(* Init ST03_125_F1 Absicherung Roboter iO (DigIn) *)
ST03_125_F1.sInit.InstName               :='ST03_125_F1';
ST03_125_F1.sInit.Description            :='Absicherung Roboter iO';
ST03_125_F1.sInit.BitInName              :='+3-125_F1';
ST03_125_F1.sInit.HomePosSignal          :=2; (* 0: Signal=Low, 1: Signal=High, 2: always  *)
ST03_125_F1.sInit.MaxTime                :=10;
ST03_125_F1.sInit.EnableInEveryMode       :=TRUE;

(* Init ST03_400_B12_6 Schwenkmodul GST (Roboterkopf) (DigIn) *)
ST03_400_B12_6.sInit.InstName           :='ST03_400_B12_6';
ST03_400_B12_6.sInit.Description        :='Rob. ST03 Schwenken GST';
ST03_400_B12_6.sInit.BitInName          :='+3-400_B12_6';
ST03_400_B12_6.sInit.HomePosSignal      :=2; (* 0: Signal=Low, 1: Signal=High, 2: always  *)
ST03_400_B12_6.sInit.MaxTime            :=2000;

(* Init ST03_400_B12_7 Schwenkmodul AST (Roboter) (DigIn) *)
ST03_400_B12_7.sInit.InstName           :='ST03_400_B12_7';
ST03_400_B12_7.sInit.Description        :='Rob. ST03 Schwenken AST';
ST03_400_B12_7.sInit.BitInName          :='+3-400_B12_7';
ST03_400_B12_7.sInit.HomePosSignal      :=2; (* 0: Signal=Low, 1: Signal=High, 2: always  *)
ST03_400_B12_7.sInit.MaxTime            :=2000;

(* Init St03_120_A1_A14 Rob. opt. Tool 2 ist Ein (DigIn) *)
St03_120_A1_A14.sInit.InstName           :='St03_120_A1_A14';
St03_120_A1_A14.sInit.Description        :='Rob. opt. Tool 2 ist Ein';
St03_120_A1_A14.sInit.BitInName          :='+3-120_A1_A14';
St03_120_A1_A14.sInit.HomePosSignal      :=2; (* 0: Signal=Low, 1: Signal=High, 2: always  *)
St03_120_A1_A14.sInit.MaxTime            :=2000;

(* Init ST03_BG3_S53_0 Start Band für Dummyprüfung (DigIn) *)
ST03_BG3_S53_0.sInit.InstName               :='ST03_BG3_S53_0';
ST03_BG3_S53_0.sInit.Description            :='Start Band für Dummyprüfung';
ST03_BG3_S53_0.sInit.BitInName              :='+0-BG3_S53_0';
ST03_BG3_S53_0.sInit.HomePosSignal          :=2; (* 0: Signal=Low, 1: Signal=High, 2: always  *)
ST03_BG3_S53_0.sInit.MaxTime                :=2000;
ST03_BG3_S53_0.sInit.EnableInEveryMode   	 :=TRUE;

(* Init ST03_BG3_X53_0 LED TasterStart Band für Dummyprüfung (DigOutIn) *)
ST03_BG3_X53_0.sInit.InstName          :='ST03_BG3_X53_0';
ST03_BG3_X53_0.sInit.Description       :='LED TasterStart Band für Dummyprüfung';
ST03_BG3_X53_0.sInit.BitOutName        :='+ST03_BG3_X53_0';
ST03_BG3_X53_0.sInit.BitInName         :='';
ST03_BG3_X53_0.sInit.HomePosSignal     :=2; (* 0: Signal=Low, 1: Signal=High, 2: always  *)
ST03_BG3_X53_0.sInit.MaxTime           :=2000;

(* Init ST03_400_B54_7 Tray Testteile in Position (DigIn) *)
ST03_400_B54_7.sInit.InstName            :='ST03_400_B54_7';
ST03_400_B54_7.sInit.Description         :='Tray Testteile in Position';
ST03_400_B54_7.sInit.BitInName           :='+8-400_B54.7';
ST03_400_B54_7.sInit.HomePosSignal       :=2; (* 0: Signal=Low, 1: Signal=High, 2: always  *)
ST03_400_B54_7.sInit.MaxTime             :=2000;

(* Init ST03_8_75_B13_5 voll/belegt keine Prüfteile mehr (DigIn) *)
ST03_8_75_B13_5.sInit.InstName            :='ST03_8_75_B13_5';
ST03_8_75_B13_5.sInit.Description         :='voll/belegt keine Prüfteile mehr';
ST03_8_75_B13_5.sInit.BitInName           :='+8-75_B13.5';
ST03_8_75_B13_5.sInit.HomePosSignal       :=2; (* 0: Signal=Low, 1: Signal=High, 2: always  *)
ST03_8_75_B13_5.sInit.MaxTime             :=2000;

(* Init ST03_8_75_B13_6 belegt mit 6 Prüfteile (DigIn) *)
ST03_8_75_B13_6.sInit.InstName            :='ST03_8_75_B13_6';
ST03_8_75_B13_6.sInit.Description         :='belegt mit 6 Prüfteile';
ST03_8_75_B13_6.sInit.BitInName           :='+8-75_B13.6';
ST03_8_75_B13_6.sInit.HomePosSignal       :=2; (* 0: Signal=Low, 1: Signal=High, 2: always  *)
ST03_8_75_B13_6.sInit.MaxTime             :=2000;

(* Init ST03_65_Q1 LED TasterStart Band für Dummyprüfung (DigOutIn) *)
ST03_65_Q1.sInit.InstName          :='ST03_65_Q1';
ST03_65_Q1.sInit.Description       :='Kühltunnel (Lüfter)';
ST03_65_Q1.sInit.BitOutName        :='+ST03_65_Q1';
ST03_65_Q1.sInit.BitInName         :='';
ST03_65_Q1.sInit.HomePosSignal     :=2; (* 0: Signal=Low, 1: Signal=High, 2: always  *)
ST03_65_Q1.sInit.MaxTime           :=2000;

(* Init ST03_65_F1 Tray Testteile in Position (DigIn) *)
ST03_65_F1.sInit.InstName            :='ST03_65_F1';
ST03_65_F1.sInit.Description         :='Sicherung Kühltunnel (Lüfter)';
ST03_65_F1.sInit.BitInName           :='+8-65_F1';
ST03_65_F1.sInit.HomePosSignal       :=2; (* 0: Signal=Low, 1: Signal=High, 2: always  *)
ST03_65_F1.sInit.MaxTime             :=2000;
END_PROGRAM
ACTION Init_120pol:
(*Rüstsatz 120 pol ==================================================================================*)

(* Init ST03_531_B69_0 Zuführung  frei zum Ablegen ISK SP Maschine (DigIn) *)
ST03_531_B69_0.sInit.InstName            :='ST03_531_B69_0';
ST03_531_B69_0.sInit.Description         :='frei zum Ablegen ISK SP Maschine';
ST03_531_B69_0.sInit.BitInName           :='+8-531_B69.0';
ST03_531_B69_0.sInit.HomePosSignal       :=2; (* 0: Signal=Low, 1: Signal=High, 2: always  *)
ST03_531_B69_0.sInit.MaxTime             :=2000;
ST03_531_B69_0.sInit.EnableInEveryMode   :=TRUE;

(* Init ST03_531_B69_1 Zuführung Vereinzler eingefahren GST (ValveSensor) *)
ST03_531_B69_1.sInit.InstName		:='ST03_531_B69_1';
ST03_531_B69_1.sInit.BitName		:='+8_531_B69.1';
ST03_531_B69_1.sInit.Description	:=' Vereinzler eingefahren GST';
ST03_531_B69_1.sInit.SensorType	:=sValveSensorType_INIT;

(* Init ST03_531_B69_2 Zuführung Vereinzler ausgefahren AST (ValveSensor) *)
ST03_531_B69_2.sInit.InstName		:='ST03_531_B69_2';
ST03_531_B69_2.sInit.BitName		:='+8_531_B69.2';
ST03_531_B69_2.sInit.Description	:=' Vereinzler ausgefahren AST';
ST03_531_B69_2.sInit.SensorType	:=sValveSensorType_WORK;

(* Init ST03_531_B69_3 Zuführung Stopper eingefahren AST (ValveSensor) *)
ST03_531_B69_3.sInit.InstName		:='ST03_531_B69_3';
ST03_531_B69_3.sInit.BitName		:='+8_531_B69.3';
ST03_531_B69_3.sInit.Description	:='Stopper eingefahren AST';
ST03_531_B69_3.sInit.SensorType	:=sValveSensorType_WORK;

(* Init ST03_531_B69_4 Zuführung Stopper ausgefahren GST (ValveSensor) *)
ST03_531_B69_4.sInit.InstName		:='ST03_531_B69_4';
ST03_531_B69_4.sInit.BitName		:='+8_531_B69.4';
ST03_531_B69_4.sInit.Description	:='Stopper ausgefahren GST';
ST03_531_B69_4.sInit.SensorType	:=sValveSensorType_INIT;;

(* Init ST03_531_B69_6 ISK anwesend am Stopper (DigIn) *)
ST03_531_B69_6.sInit.InstName            :='ST03_531_B69_6';
ST03_531_B69_6.sInit.Description         :='ISK anwesend am Stopper';
ST03_531_B69_6.sInit.BitInName           :='+8-531_B69.6';
ST03_531_B69_6.sInit.HomePosSignal       :=2; (* 0: Signal=Low, 1: Signal=High, 2: always  *)
ST03_531_B69_6.sInit.MaxTime             :=2000;
ST03_531_B69_6.sInit.EnableInEveryMode   :=TRUE;

(* Init ST03_531_B69_7 ISK rechts Lageerkennung (DigIn) *)
ST03_531_B69_7.sInit.InstName            :='ST03_531_B69_7';
ST03_531_B69_7.sInit.Description         :='ISK Lageerkennung rechts.';
ST03_531_B69_7.sInit.BitInName           :='+8-531_B69.7';
ST03_531_B69_7.sInit.HomePosSignal       :=2; (* 0: Signal=Low, 1: Signal=High, 2: always  *)
ST03_531_B69_7.sInit.MaxTime             :=2000;
ST03_531_B69_7.sInit.EnableInEveryMode   :=TRUE;

(* Init ST03_562_B70_0 ISK links Lageerkennung (DigIn) *)
ST03_532_B70_0.sInit.InstName            :='ST03_532_B70_0';
ST03_532_B70_0.sInit.Description         :='ISK Lageerkennung links';
ST03_532_B70_0.sInit.BitInName           :='+8-532_B70.0';
ST03_532_B70_0.sInit.HomePosSignal       :=2; (* 0: Signal=Low, 1: Signal=High, 2: always  *)
ST03_532_B70_0.sInit.MaxTime             :=2000;
ST03_532_B70_0.sInit.EnableInEveryMode   :=TRUE;

(* Init ST03_532_Y70_1   Zuführung  Vereinzler AST/GST (Valve) *)
ST03_532_Y70_1.sInit.InstName            :='ST03_532_Y70_1';
ST03_532_Y70_1.sInit.BitName            :='+8-532_Y70.1';
ST03_532_Y70_1.sInit.Description         :=' Zuführung Vereinzler AST/GST';
ST03_532_Y70_1.sInit.HomePosDefine       :=HOME_ALWAYS;
ST03_532_Y70_1.sInit.InitDescription     :='GS einfahren';
ST03_532_Y70_1.sInit.WorkDescription     :='AS ausfahren';
ST03_532_Y70_1.sInit.DampBothTime        :=200;
ST03_532_Y70_1.sInit.KindOfValve         :='A';
ST03_532_Y70_1.sInit.MaxTime             :=2000;

(* Init ST03_532_Y70_2   Zuführung  Stopper AST/GST (Valve) *)
ST03_532_Y70_2.sInit.InstName            :='ST03_532_Y70_2';
ST03_532_Y70_2.sInit.BitName            :='+8-532_Y70.2';
ST03_532_Y70_2.sInit.Description         :=' Zuführung Stopper AST/GST';
ST03_532_Y70_2.sInit.HomePosDefine       :=HOME_ALWAYS;
ST03_532_Y70_2.sInit.InitDescription     :='GS ausfahren';
ST03_532_Y70_2.sInit.WorkDescription     :='AS einfahren';
ST03_532_Y70_2.sInit.DampBothTime        :=200;
ST03_532_Y70_2.sInit.KindOfValve         :='A';
ST03_532_Y70_2.sInit.MaxTime             :=2000;
END_ACTION
ACTION Init_124pol:
(*========================= Rüstsatz 124 polig===============================*)

(* Init ST03_451_B69_0 Förderbandeinheit  Zuführung Vereinzler AST (ValveSensor) *)
ST03_451_B69_0.sInit.InstName            :='ST03_451_B69_0';
ST03_451_B69_0.sInit.BitName            :='+8_451_B69.0';
ST03_451_B69_0.sInit.Description         :='Förderbandeinheit  Zuführung Vereinzler AST';
ST03_451_B69_0.sInit.SensorType          :=sValveSensorType_INIT;

(* Init ST03_451_B69_1 Förderbandeinheit  Zuführung Vereinzler GST (ValveSensor) *)
ST03_451_B69_1.sInit.InstName            :='ST03_451_B69_1';
ST03_451_B69_1.sInit.BitName            :='+8_451_B69.1';
ST03_451_B69_1.sInit.Description         :='Förderbandeinheit  Zuführung Vereinzler GST';
ST03_451_B69_1.sInit.SensorType          :=sValveSensorType_WORK;

(* Init ST03_451_B69_2 Förderbandeinheit  Zuführung Stopper AST (ValveSensor) *)
ST03_451_B69_2.sInit.InstName            :='ST03_451_B69_2';
ST03_451_B69_2.sInit.BitName            :='+8_451_B69.2';
ST03_451_B69_2.sInit.Description         :='Förderband linke Zuführung Stopper AST';
ST03_451_B69_2.sInit.SensorType          :=sValveSensorType_INIT;

(* Init ST03_451_B69_3 Förderbandeinheit  Zuführung Stopper GST (ValveSensor) *)
ST03_451_B69_3.sInit.InstName            :='ST03_451_B69_3';
ST03_451_B69_3.sInit.BitName            :='+8_451_B69.3';
ST03_451_B69_3.sInit.Description         :='Förderband linke Zuführung Stopper GST';
ST03_451_B69_3.sInit.SensorType          :=sValveSensorType_WORK;

(* Init ST03_451_B69_4  Zuführung  frei zum Ablegen ISK SP Maschine Pos.1 (DigIn) *)
ST03_451_B69_4.sInit.InstName            :='ST03_451_B69_4';
ST03_451_B69_4.sInit.Description         :='Zuführung links frei zum Ablegen ISK SP Maschine Pos1';
ST03_451_B69_4.sInit.BitInName           :='+8-451_B69.4';
ST03_451_B69_4.sInit.HomePosSignal       :=2; (* 0: Signal=Low, 1: Signal=High, 2: always  *)
ST03_451_B69_4.sInit.MaxTime             :=2000;
ST03_451_B69_4.sInit.EnableInEveryMode   :=TRUE;

(* Init ST03_451_B69_7  ISK anwesend am Vereinzler (DigIn) *)
ST03_451_B69_7.sInit.InstName            :='ST03_451_B69_7';
ST03_451_B69_7.sInit.Description         :='ISK anwesend am Vereinzler';
ST03_451_B69_7.sInit.BitInName           :='+8-451_B69.7';
ST03_451_B69_7.sInit.HomePosSignal       :=2; (* 0: Signal=Low, 1: Signal=High, 2: always  *)
ST03_451_B69_7.sInit.MaxTime             :=2000;
ST03_451_B69_7.sInit.EnableInEveryMode   :=TRUE;

(* Init ST03_452_B70_1  Züführung  ISK Lageerkennung 1 (DigIn) *)
ST03_452_B70_1.sInit.InstName            :='ST03_452_B70_1';
ST03_452_B70_1.sInit.Description         :='Züführung  ISK Lageerkennung 1';
ST03_452_B70_1.sInit.BitInName           :='+8-452_B70.1';
ST03_452_B70_1.sInit.HomePosSignal       :=2; (* 0: Signal=Low, 1: Signal=High, 2: always  *)
ST03_452_B70_1.sInit.MaxTime             :=2000;
ST03_452_B70_1.sInit.EnableInEveryMode   :=TRUE;

(* Init ST03_452_B70_2  Züführung  ISK Lageerkennung 2 (DigIn) *)
ST03_452_B70_2.sInit.InstName            :='ST03_452_B70_2';
ST03_452_B70_2.sInit.Description         :='Züführung  ISK Lageerkennung 2';
ST03_452_B70_2.sInit.BitInName           :='+8-452_B70.2';
ST03_452_B70_2.sInit.HomePosSignal       :=2; (* 0: Signal=Low, 1: Signal=High, 2: always  *)
ST03_452_B70_2.sInit.MaxTime             :=2000;
ST03_452_B70_2.sInit.EnableInEveryMode   :=TRUE;

(* Init ST03_453_B70_4  ISK anwesend Übergabeposition Roboter (DigIn) *)
ST03_453_B70_4.sInit.InstName            :='ST03_453_B70_4';
ST03_453_B70_4.sInit.Description         :='Zuführung ISK auf Übergabeposition Robo Palettierer ';
ST03_453_B70_4.sInit.BitInName           :='+8-453_B70.4';
ST03_453_B70_4.sInit.HomePosSignal       :=2; (* 0: Signal=Low, 1: Signal=High, 2: always  *)
ST03_453_B70_4.sInit.MaxTime             :=2000;
ST03_453_B70_4.sInit.EnableInEveryMode   :=TRUE;

(* Init ST03_453_Y70_5 Förderband  Zuführung Vereinzler (Valve) *)
ST03_453_Y70_5.sInit.InstName            :='ST03_453_Y70_5';
ST03_453_Y70_5.sInit.BitName            :='+8-453_Y70.5';
ST03_453_Y70_5.sInit.Description         :='Förderband  Zuführung Vereinzler';
ST03_453_Y70_5.sInit.HomePosDefine       :=HOME_ALWAYS;
ST03_453_Y70_5.sInit.InitDescription     :='GS einfahren';
ST03_453_Y70_5.sInit.WorkDescription     :='AS ausfahren';
ST03_453_Y70_5.sInit.DampBothTime        :=200;
ST03_453_Y70_5.sInit.KindOfValve         :='A';
ST03_453_Y70_5.sInit.MaxTime             :=2000;

(* Init ST03_453_Y70_6 Förderband  Zuführung Stopper (Valve) *)
ST03_453_Y70_6.sInit.InstName            :='ST03_453_Y70_6';
ST03_453_Y70_6.sInit.BitName            :='+8-453_Y70.6';
ST03_453_Y70_6.sInit.Description         :='Förderband  Zuführung Stopper';
ST03_453_Y70_6.sInit.HomePosDefine       :=HOME_ALWAYS;
ST03_453_Y70_6.sInit.InitDescription     :='GS ausfahren';
ST03_453_Y70_6.sInit.WorkDescription     :='AS einfahren';
ST03_453_Y70_6.sInit.DampBothTime        :=200;
ST03_453_Y70_6.sInit.KindOfValve         :='A';
ST03_453_Y70_6.sInit.MaxTime             :=2000;
END_ACTION
ACTION Init_154pol:
(*Rüstsatz 154pol*)
(* Init ST03_425_B67_0 Förderbandeinheit  Zuführung Vereinzler AST (ValveSensor) *)
ST03_425_B67_0.sInit.InstName            :='ST03_425_B67_0';
ST03_425_B67_0.sInit.BitName            :='+8_425_B67.0';
ST03_425_B67_0.sInit.Description         :='Förderbandeinheit  Zuführung Vereinzler AST';
ST03_425_B67_0.sInit.SensorType          :=sValveSensorType_INIT;

(* Init ST03_425_B67_1 Förderbandeinheit  Zuführung Vereinzler GST (ValveSensor) *)
ST03_425_B67_1.sInit.InstName            :='ST03_425_B67_1';
ST03_425_B67_1.sInit.BitName            :='+8_425_B67.1';
ST03_425_B67_1.sInit.Description         :='Förderbandeinheit  Zuführung Vereinzler GST';
ST03_425_B67_1.sInit.SensorType          :=sValveSensorType_WORK;

(* Init ST03_425_B67_2 Förderbandeinheit  Zuführung Stopper AST (ValveSensor) *)
ST03_425_B67_2.sInit.InstName            :='ST03_425_B67_2';
ST03_425_B67_2.sInit.BitName            :='+8_425_B67.2';
ST03_425_B67_2.sInit.Description         :='Förderband linke Zuführung Stopper AST';
ST03_425_B67_2.sInit.SensorType          :=sValveSensorType_INIT;

(* Init ST03_425_B67_3 Förderbandeinheit  Zuführung Stopper GST (ValveSensor) *)
ST03_425_B67_3.sInit.InstName            :='ST03_425_B67_3';
ST03_425_B67_3.sInit.BitName            :='+8_425_B67.3';
ST03_425_B67_3.sInit.Description         :='Förderband linke Zuführung Stopper GST';
ST03_425_B67_3.sInit.SensorType          :=sValveSensorType_WORK;

(* Init ST03_425_B67_4  Zuführung  frei zum Ablegen ISK SP Maschine Pos.1 (DigIn) *)
ST03_425_B67_4.sInit.InstName            :='ST03_425_B67_4';
ST03_425_B67_4.sInit.Description         :='Zuführung links frei zum Ablegen ISK SP Maschine Pos1';
ST03_425_B67_4.sInit.BitInName           :='+8-425_B67.4';
ST03_425_B67_4.sInit.HomePosSignal       :=2; (* 0: Signal=Low, 1: Signal=High, 2: always  *)
ST03_425_B67_4.sInit.MaxTime             :=2000;
ST03_425_B67_4.sInit.EnableInEveryMode   :=TRUE;

(* Init ST03_425_B67_5  Zuführung  frei zum Ablegen ISK SP Maschine Pos.2 (DigIn) *)
ST03_425_B67_5.sInit.InstName            :='ST03_425_B67_5';
ST03_425_B67_5.sInit.Description         :='Zuführung links frei zum Ablegen ISK SP Maschine Pos2';
ST03_425_B67_5.sInit.BitInName           :='+8-425_B67.5';
ST03_425_B67_5.sInit.HomePosSignal       :=2; (* 0: Signal=Low, 1: Signal=High, 2: always  *)
ST03_425_B67_5.sInit.MaxTime             :=2000;
ST03_425_B67_5.sInit.EnableInEveryMode   :=TRUE;

(* Init ST03_425_B67_6  Zuführung  frei zum Ablegen ISK SP Maschine Pos.3 (DigIn) *)
ST03_425_B67_6.sInit.InstName            :='ST03_425_B67_6';
ST03_425_B67_6.sInit.Description         :='Zuführung links frei zum Ablegen ISK SP Maschine Pos3';
ST03_425_B67_6.sInit.BitInName           :='+8-425_B67.6';
ST03_425_B67_6.sInit.HomePosSignal       :=2; (* 0: Signal=Low, 1: Signal=High, 2: always  *)
ST03_425_B67_6.sInit.MaxTime             :=2000;
ST03_425_B67_6.sInit.EnableInEveryMode   :=TRUE;

(* Init ST03_425_B67_7  ISK anwesend am Vereinzler (DigIn) *)
ST03_425_B67_7.sInit.InstName            :='ST03_425_B67_7';
ST03_425_B67_7.sInit.Description         :='ISK anwesend am Vereinzler';
ST03_425_B67_7.sInit.BitInName           :='+8-425_B67.7';
ST03_425_B67_7.sInit.HomePosSignal       :=2; (* 0: Signal=Low, 1: Signal=High, 2: always  *)
ST03_425_B67_7.sInit.MaxTime             :=2000;
ST03_425_B67_7.sInit.EnableInEveryMode   :=TRUE;

(* Init ST03_426_B68_4  Züführung  ISK auf Übergabeposition Roboter Palettierer (DigIn) *)
ST03_426_B68_4.sInit.InstName            :='ST03_426_B68_4';
ST03_426_B68_4.sInit.Description         :='Züführung  ISK auf Übergabeposition Roboter Palettierer';
ST03_426_B68_4.sInit.BitInName           :='+8-426_B68.4';
ST03_426_B68_4.sInit.HomePosSignal       :=2; (* 0: Signal=Low, 1: Signal=High, 2: always  *)
ST03_426_B68_4.sInit.MaxTime             :=2000;
ST03_426_B68_4.sInit.EnableInEveryMode   :=TRUE;

(* Init ST03_426_Y68_5 Förderband  Zuführung Vereinzler (Valve) *)
ST03_426_Y68_5.sInit.InstName            :='ST03_426_Y68_5';
ST03_426_Y68_5.sInit.BitName            :='+8-426_Y68.5';
ST03_426_Y68_5.sInit.Description         :='Förderband  Zuführung Vereinzler';
ST03_426_Y68_5.sInit.HomePosDefine       :=HOME_ALWAYS;
ST03_426_Y68_5.sInit.InitDescription     :='GS einfahren';
ST03_426_Y68_5.sInit.WorkDescription     :='AS ausfahren';
ST03_426_Y68_5.sInit.DampBothTime        :=200;
ST03_426_Y68_5.sInit.KindOfValve         :='A';
ST03_426_Y68_5.sInit.MaxTime             :=2000;

(* Init ST03_426_Y68_6 Förderband  Zuführung Stopper (Valve) *)
ST03_426_Y68_6.sInit.InstName            :='ST03_426_Y68_6';
ST03_426_Y68_6.sInit.BitName            :='+8-426_Y68.6';
ST03_426_Y68_6.sInit.Description         :='Förderband  Zuführung Stopper';
ST03_426_Y68_6.sInit.HomePosDefine       :=HOME_ALWAYS;
ST03_426_Y68_6.sInit.InitDescription     :='GS ausfahren';
ST03_426_Y68_6.sInit.WorkDescription     :='AS einfahren';
ST03_426_Y68_6.sInit.DampBothTime        :=200;
ST03_426_Y68_6.sInit.KindOfValve         :='A';
ST03_426_Y68_6.sInit.MaxTime             :=2000;
END_ACTION
ACTION Init_154polRP:
(*Rüstsatz 154 Rasterplattel*)

(* Init ST03_418_B60_0 Förderband linke Zuführung Vereinzler AST  (ValveSensor) *)
ST03_418_B60_0.sInit.InstName            :='ST03_418_B60_0';
ST03_418_B60_0.sInit.BitName            :='+8_418_B60.0';
ST03_418_B60_0.sInit.Description         :='Förderband linke Zuführung Vereinzler AST';
ST03_418_B60_0.sInit.SensorType          :=sValveSensorType_WORK;

(* Init ST03_418_B60_1 Förderband linke Zuführung Vereinzler GST (ValveSensor) *)
ST03_418_B60_1.sInit.InstName            :='ST03_418_B60_1';
ST03_418_B60_1.sInit.BitName            :='+8_418_B60.1';
ST03_418_B60_1.sInit.Description         :='Förderband linke Zuführung Vereinzler GST';
ST03_418_B60_1.sInit.SensorType          :=sValveSensorType_INIT;

(* Init ST03_418_B60_2 Förderband rechte Zuführung Vereinzler AST (ValveSensor) *)
ST03_418_B60_2.sInit.InstName            :='ST03_418_B60_2';
ST03_418_B60_2.sInit.BitName            :='+8_418_B60.2';
ST03_418_B60_2.sInit.Description         :='Förderband rechte Zuführung Vereinzler AST';
ST03_418_B60_2.sInit.SensorType          :=sValveSensorType_WORK;

(* Init ST03_418_B60_3 Förderband rechte Zuführung Vereinzler GST(ValveSensor) *)
ST03_418_B60_3.sInit.InstName            :='ST03_418_B60_3';
ST03_418_B60_3.sInit.BitName            :='+8_418_B60.3';
ST03_418_B60_3.sInit.Description         :=' Förderband rechte Zuführung Vereinzler GST';
ST03_418_B60_3.sInit.SensorType          :=sValveSensorType_INIT;

(* Init ST03_418_B60_4 Förderband links/rechts Zuführung Stopper AST (ValveSensor) *)
ST03_418_B60_4.sInit.InstName            :='ST03_418_B60_4';
ST03_418_B60_4.sInit.BitName            :='+8_418_B60.4';
ST03_418_B60_4.sInit.Description         :='Förderband links/rechts Zuführung Stopper AST';
ST03_418_B60_4.sInit.SensorType          :=sValveSensorType_WORK;

(* Init ST03_418_B60_5 Förderband links/rechts Zuführung Stopper GST (ValveSensor) *)
ST03_418_B60_5.sInit.InstName            :='ST03_418_B60_5';
ST03_418_B60_5.sInit.BitName            :='+8_418_B60.5';
ST03_418_B60_5.sInit.Description         :='Förderband links/rechts Zuführung Stopper GST';
ST03_418_B60_5.sInit.SensorType          :=sValveSensorType_INIT;

(* Init ST03_418_B60_6 Zuführung links frei zum Ablegen ISK SP Maschine (DigIn) *)
ST03_418_B60_6.sInit.InstName            :='ST03_418_B60_6';
ST03_418_B60_6.sInit.Description         :='Zuführung links frei zum Ablegen ISK SP Maschine';
ST03_418_B60_6.sInit.BitInName           :='+8-418_B60.6';
ST03_418_B60_6.sInit.HomePosSignal       :=2; (* 0: Signal=Low, 1: Signal=High, 2: always  *)
ST03_418_B60_6.sInit.MaxTime             :=2000;
ST03_418_B60_6.sInit.EnableInEveryMode   :=TRUE;

(* Init ST03_418_B60_7 Zuführung rechts frei zum Ablegen ISK SP Maschine (DigIn) *)
ST03_418_B60_7.sInit.InstName            :='ST03_418_B60_7';
ST03_418_B60_7.sInit.Description         :='Zuführung rechts frei zum Ablegen ISK SP Maschine';
ST03_418_B60_7.sInit.BitInName           :='+8-418_B60.7';
ST03_418_B60_7.sInit.HomePosSignal       :=2; (* 0: Signal=Low, 1: Signal=High, 2: always  *)
ST03_418_B60_7.sInit.MaxTime             :=2000;
ST03_418_B60_7.sInit.EnableInEveryMode   :=TRUE;

(* Init ST03_419_B61_0 Förderband Zuführung links ISK anwesend zum Vereinzeln (DigIn) *)
ST03_419_B61_0.sInit.InstName            :='ST03_419_B61_0';
ST03_419_B61_0.sInit.Description         :='Förderband Zuführung links ISK anwesend zum Vereinzeln';
ST03_419_B61_0.sInit.BitInName           :='+8-419_B61.0';
ST03_419_B61_0.sInit.HomePosSignal       :=2; (* 0: Signal=Low, 1: Signal=High, 2: always  *)
ST03_419_B61_0.sInit.MaxTime             :=2000;
ST03_419_B61_0.sInit.EnableInEveryMode   :=TRUE;

(* Init ST03_419_B61_1 Förderband Zuführung rechts ISK anwesend zum Vereinzeln (DigIn) *)
ST03_419_B61_1.sInit.InstName            :='ST03_419_B61_1';
ST03_419_B61_1.sInit.Description         :='Förderband Zuführung rechts ISK anwesend zum Vereinzeln';
ST03_419_B61_1.sInit.BitInName           :='+8-419_B61.1';
ST03_419_B61_1.sInit.HomePosSignal       :=2; (* 0: Signal=Low, 1: Signal=High, 2: always  *)
ST03_419_B61_1.sInit.MaxTime             :=2000;
ST03_419_B61_1.sInit.EnableInEveryMode   :=TRUE;

(* Init ST03_419_B61_2 Züführung links ISK auf Übergabeposition Roboter Palettierer (DigIn) *)
ST03_419_B61_2.sInit.InstName            :='ST03_419_B61_2';
ST03_419_B61_2.sInit.Description         :='Züführung links ISK auf Übergabeposition Roboter Palettierer';
ST03_419_B61_2.sInit.BitInName           :='+8-419_B61.2';
ST03_419_B61_2.sInit.HomePosSignal       :=2; (* 0: Signal=Low, 1: Signal=High, 2: always  *)
ST03_419_B61_2.sInit.MaxTime             :=2000;
ST03_419_B61_2.sInit.EnableInEveryMode   :=TRUE;

(* Init ST03_419_B61_3 Züführung rechts ISK auf Übergabeposition Roboter Palettierer (DigIn) *)
ST03_419_B61_3.sInit.InstName            :='ST03_419_B61_3';
ST03_419_B61_3.sInit.Description         :='Züführung rechts ISK auf Übergabeposition Roboter Palettierer';
ST03_419_B61_3.sInit.BitInName           :='+8-419_B61.3';
ST03_419_B61_3.sInit.HomePosSignal       :=2; (* 0: Signal=Low, 1: Signal=High, 2: always  *)
ST03_419_B61_3.sInit.MaxTime             :=2000;
ST03_419_B61_3.sInit.EnableInEveryMode   :=TRUE;

(* Init ST03_419_Y61_5 Förderband linke Zuführung Vereinzler AST/GST (Valve) *)
ST03_419_Y61_5.sInit.InstName            :='ST03_419_Y61_5';
ST03_419_Y61_5.sInit.BitName            :='+8-419_Y61.5';
ST03_419_Y61_5.sInit.Description         :='Förderband linke Zuführung Vereinzler AST/GST';
ST03_419_Y61_5.sInit.HomePosDefine       :=HOME_ALWAYS;
ST03_419_Y61_5.sInit.InitDescription     :='GS einfahren';
ST03_419_Y61_5.sInit.WorkDescription     :='AS ausfahren';
ST03_419_Y61_5.sInit.DampBothTime        :=200;
ST03_419_Y61_5.sInit.KindOfValve         :='A';
ST03_419_Y61_5.sInit.MaxTime             :=2000;

(* Init ST03_419_Y61_6 Förderband rechte Zuführung Vereinzler AST/GST (Valve) *)
ST03_419_Y61_6.sInit.InstName            :='ST03_419_Y61_6';
ST03_419_Y61_6.sInit.BitName            :='+8-419_Y61.6';
ST03_419_Y61_6.sInit.Description         :='Förderband rechte Zuführung Vereinzler AST/GST';
ST03_419_Y61_6.sInit.HomePosDefine       :=HOME_ALWAYS;
ST03_419_Y61_6.sInit.InitDescription     :='GS einfahren';
ST03_419_Y61_6.sInit.WorkDescription     :='AS ausfahren';
ST03_419_Y61_6.sInit.DampBothTime        :=200;
ST03_419_Y61_6.sInit.KindOfValve         :='A';
ST03_419_Y61_6.sInit.MaxTime             :=2000;

(* Init ST03_419_Y61_7 Förderband links/rechts Züführung Stopper AST/GST (Valve) *)
ST03_419_Y61_7.sInit.InstName            :='ST03_419_Y61_7';
ST03_419_Y61_7.sInit.BitName            :='+8-419_Y61.7';
ST03_419_Y61_7.sInit.Description         :='Förderband links/rechts Züführung Stopper AST/GST';
ST03_419_Y61_7.sInit.HomePosDefine       :=HOME_ALWAYS;
ST03_419_Y61_7.sInit.InitDescription     :='GS ausfahren';
ST03_419_Y61_7.sInit.WorkDescription     :='AS einfahren';
ST03_419_Y61_7.sInit.DampBothTime        :=200;
ST03_419_Y61_7.sInit.KindOfValve         :='A';
ST03_419_Y61_7.sInit.MaxTime             :=2000;
END_ACTION
ACTION Init_160pol:
(*Rüstsatz 160pol*)
(* Init ST03_421_B63_0  Förderband Zuführung Vereinzler AST  (ValveSensor) *)
ST03_421_B63_0.sInit.InstName            :='ST03_421_B63_0';
ST03_421_B63_0.sInit.BitName            :='+8_421_B63.0';
ST03_421_B63_0.sInit.Description         :=' Förderband Zuführung Vereinzler AST';
ST03_421_B63_0.sInit.SensorType          :=sValveSensorType_WORK;

(* Init ST03_421_B63_1  Förderband Zuführung Vereinzler GST  (ValveSensor) *)
ST03_421_B63_1.sInit.InstName            :='ST03_421_B63_1';
ST03_421_B63_1.sInit.BitName            :='+8_421_B63.1';
ST03_421_B63_1.sInit.Description         :=' Förderband Zuführung Vereinzler GST';
ST03_421_B63_1.sInit.SensorType          :=sValveSensorType_INIT;

(* Init ST03_421_B63_2  Förderband Zuführung Stopper AST  (ValveSensor) *)
ST03_421_B63_2.sInit.InstName            :='ST03_421_B63_2';
ST03_421_B63_2.sInit.BitName            :='+8_421_B63.2';
ST03_421_B63_2.sInit.Description         :=' Förderband Zuführung Stopper AST';
ST03_421_B63_2.sInit.SensorType          :=sValveSensorType_INIT;

(* Init ST03_421_B63_3  Förderband Zuführung Stopper GST  (ValveSensor) *)
ST03_421_B63_3.sInit.InstName            :='ST03_421_B63_3';
ST03_421_B63_3.sInit.BitName            :='+8_421_B63.3';
ST03_421_B63_3.sInit.Description         :=' Förderband Zuführung Stopper GST';
ST03_421_B63_3.sInit.SensorType          :=sValveSensorType_WORK;

(* Init ST03_421_B63_4 Förderband frei zum Ablegen ISK SP Maschine Pos1 (DigIn) *)
ST03_421_B63_4.sInit.InstName            :='ST03_421_B63_4';
ST03_421_B63_4.sInit.Description         :='Förderband frei zum Ablegen ISK SP Maschine Pos1';
ST03_421_B63_4.sInit.BitInName           :='+8-421_B63.4';
ST03_421_B63_4.sInit.HomePosSignal       :=2; (* 0: Signal=Low, 1: Signal=High, 2: always  *)
ST03_421_B63_4.sInit.MaxTime             :=2000;
ST03_421_B63_4.sInit.EnableInEveryMode   :=TRUE;

(* Init ST03_421_B63_5 Förderband frei zum Ablegen ISK SP Maschine Pos2 (DigIn) *)
ST03_421_B63_5.sInit.InstName            :='ST03_421_B63_5';
ST03_421_B63_5.sInit.Description         :='Förderband frei zum Ablegen ISK SP Maschine Pos2';
ST03_421_B63_5.sInit.BitInName           :='+8-421_B63.5';
ST03_421_B63_5.sInit.HomePosSignal       :=2; (* 0: Signal=Low, 1: Signal=High, 2: always  *)
ST03_421_B63_5.sInit.MaxTime             :=2000;
ST03_421_B63_5.sInit.EnableInEveryMode   :=TRUE;

(* Init ST03_421_B63_6 Förderband frei zum Ablegen ISK SP Maschine Pos3 (DigIn) *)
ST03_421_B63_6.sInit.InstName            :='ST03_421_B63_6';
ST03_421_B63_6.sInit.Description         :='Förderband frei zum Ablegen ISK SP Maschine Pos3';
ST03_421_B63_6.sInit.BitInName           :='+8-421_B63.6';
ST03_421_B63_6.sInit.HomePosSignal       :=2; (* 0: Signal=Low, 1: Signal=High, 2: always  *)
ST03_421_B63_6.sInit.MaxTime             :=2000;
ST03_421_B63_6.sInit.EnableInEveryMode   :=TRUE;

(* Init ST03_421_B63_7 ISK anwesend am Vereinzler (DigIn) *)
ST03_421_B63_7.sInit.InstName            :='ST03_421_B63_7';
ST03_421_B63_7.sInit.Description         :='ISK anwesend am Vereinzler';
ST03_421_B63_7.sInit.BitInName           :='+8-421_B63.7';
ST03_421_B63_7.sInit.HomePosSignal       :=2; (* 0: Signal=Low, 1: Signal=High, 2: always  *)
ST03_421_B63_7.sInit.MaxTime             :=2000;
ST03_421_B63_7.sInit.EnableInEveryMode   :=TRUE;

(* Init ST03_422_B64_0 Förderband Trigger Tintenstrahldrucker 1 Rüstsatz (Lichtschranke) (DigIn) *)
ST03_422_B64_0.sInit.InstName            :='ST03_421_B64_0';
ST03_422_B64_0.sInit.Description         :='Förderband Trigger Tintenstrahldrucker (Lichtschranke)';
ST03_422_B64_0.sInit.BitInName           :='+8-421_B64.0';
ST03_422_B64_0.sInit.HomePosSignal       :=2; (* 0: Signal=Low, 1: Signal=High, 2: always  *)
ST03_422_B64_0.sInit.MaxTime             :=2000;
ST03_422_B64_0.sInit.EnableInEveryMode   :=TRUE;

(* Init ST03_423_B63_0 Förderband Trigger Tintenstrahldrucker 2 Rüstsatz (Lichtschranke) (DigIn) *)
ST03_423_B66_0.sInit.InstName            :='ST03_423_B66_0';
ST03_423_B66_0.sInit.Description         :='Förderband Trigger Tintenstrahldrucker (Lichtschranke)';
ST03_423_B66_0.sInit.BitInName           :='+8-423_B66.0';
ST03_423_B66_0.sInit.HomePosSignal       :=2; (* 0: Signal=Low, 1: Signal=High, 2: always  *)
ST03_423_B66_0.sInit.MaxTime             :=2000;
ST03_423_B66_0.sInit.EnableInEveryMode   :=TRUE;

(* Init ST03_8_B76_1 Förderband Trigger Tintenstrahldrucker (Lichtschranke) (DigIn) 3621 *)
ST03_8_B76_1.sInit.InstName            :='ST03_8_B76_1';
ST03_8_B76_1.sInit.Description         :='Förderband Trigger Tintenstrahldrucker (Lichtschranke)';
ST03_8_B76_1.sInit.BitInName           :='+8-B76_1';
ST03_8_B76_1.sInit.HomePosSignal       :=2; (* 0: Signal=Low, 1: Signal=High, 2: always  *)
ST03_8_B76_1.sInit.MaxTime             :=2000;
ST03_8_B76_1.sInit.EnableInEveryMode   :=TRUE;

(* Init ST03_8_B76_2 Förderband Trigger Tintenstrahldrucker (Lichtschranke) (DigIn) 3621 *)
ST03_8_B76_2.sInit.InstName            :='ST03_8_B76_2';
ST03_8_B76_2.sInit.Description         :='Förderband Trigger Tintenstrahldrucker (Lichtschranke)';
ST03_8_B76_2.sInit.BitInName           :='+8-B76_2';
ST03_8_B76_2.sInit.HomePosSignal       :=2; (* 0: Signal=Low, 1: Signal=High, 2: always  *)
ST03_8_B76_2.sInit.MaxTime             :=2000;
ST03_8_B76_2.sInit.EnableInEveryMode   :=TRUE;

(* Init ST03_422_B64_1  Förderband Zuführung Stopper 1 Kamera AST  (ValveSensor) *)
ST03_422_B64_1.sInit.InstName            :='ST03_422_B64_1';
ST03_422_B64_1.sInit.BitName            :='+8_422_B64.1';
ST03_422_B64_1.sInit.Description         :=' Förderband Zuführung Stopper Kamera AST';
ST03_422_B64_1.sInit.SensorType          :=sValveSensorType_WORK;

(* Init ST03_422_B64_2  Förderband Zuführung Stopper 1 Kamera GST  (ValveSensor) *)
ST03_422_B64_2.sInit.InstName            :='ST03_422_B64_2';
ST03_422_B64_2.sInit.BitName            :='+8_422_B64.2';
ST03_422_B64_2.sInit.Description         :=' Förderband Zuführung Stopper 1 Kamera GST';
ST03_422_B64_2.sInit.SensorType          :=sValveSensorType_INIT;

(* Init ST03_422_B64_3  Förderband ISK anwesend am Stopper 1 Kamera (DigIn) *)
ST03_422_B64_3.sInit.InstName            :='ST03_421_B64_3';
ST03_422_B64_3.sInit.Description         :=' Förderband ISK anwesend Stopper 1 Kamera';
ST03_422_B64_3.sInit.BitInName           :='+8-421_B64.3';
ST03_422_B64_3.sInit.HomePosSignal       :=2; (* 0: Signal=Low, 1: Signal=High, 2: always  *)
ST03_422_B64_3.sInit.MaxTime             :=2000;
ST03_422_B64_3.sInit.EnableInEveryMode   :=TRUE;

(* Init ST03_423_B65_0  Förderband Zuführung Stopper 2 Kamera AST  (ValveSensor) *)
ST03_423_B65_0.sInit.InstName            :='ST03_423_B65_0';
ST03_423_B65_0.sInit.BitName            :='+8_423_B65.0';
ST03_423_B65_0.sInit.Description         :=' Förderband Zuführung Stopper 2 Kamera AST';
ST03_423_B65_0.sInit.SensorType          :=sValveSensorType_WORK;

(* Init ST03_423_B65_1  Förderband Zuführung Stopper 2 Kamera GST  (ValveSensor) *)
ST03_423_B65_1.sInit.InstName            :='ST03_423_B65_1';
ST03_423_B65_1.sInit.BitName            :='+8_423_B65.1';
ST03_423_B65_1.sInit.Description         :=' Förderband Zuführung Stopper 2 Kamera GST';
ST03_423_B65_1.sInit.SensorType          :=sValveSensorType_INIT;

(* Init ST03_423_B65_2  Förderband ISK anwesend am Stopper 2 Kamera (DigIn) *)
ST03_423_B65_2.sInit.InstName            :='ST03_423_B65_2';
ST03_423_B65_2.sInit.Description         :=' Förderband ISK anwesend Stopper Kamera';
ST03_423_B65_2.sInit.BitInName           :='+8-423_B65.2';
ST03_423_B65_2.sInit.HomePosSignal       :=2; (* 0: Signal=Low, 1: Signal=High, 2: always  *)
ST03_423_B65_2.sInit.MaxTime             :=2000;
ST03_423_B65_2.sInit.EnableInEveryMode   :=TRUE;

(* Init ST03_423_B65_3  Förderband Zuführung Stopper 3 Kamera AST  (ValveSensor) *)
ST03_423_B65_3.sInit.InstName            :='ST03_423_B65_3';
ST03_423_B65_3.sInit.BitName            :='+8_423_B65.3';
ST03_423_B65_3.sInit.Description         :=' Förderband Zuführung Stopper 3 Kamera AST';
ST03_423_B65_3.sInit.SensorType          :=sValveSensorType_WORK;

(* Init ST03_423_B65_4  Förderband Zuführung Stopper 3 Kamera GST  (ValveSensor) *)
ST03_423_B65_4.sInit.InstName            :='ST03_423_B65_4';
ST03_423_B65_4.sInit.BitName            :='+8_423_B65.4';
ST03_423_B65_4.sInit.Description         :=' Förderband Zuführung Stopper 3 Kamera GST';
ST03_423_B65_4.sInit.SensorType          :=sValveSensorType_INIT;

(* Init ST03_423_B65_5  Förderband ISK anwesend am Stopper 3 Kamera (DigIn) *)
ST03_423_B65_5.sInit.InstName            :='ST03_423_B65_5';
ST03_423_B65_5.sInit.Description         :=' Förderband ISK anwesend Stopper Kamera';
ST03_423_B65_5.sInit.BitInName           :='+8-423_B65.5';
ST03_423_B65_5.sInit.HomePosSignal       :=2; (* 0: Signal=Low, 1: Signal=High, 2: always  *)
ST03_423_B65_5.sInit.MaxTime             :=2000;
ST03_423_B65_5.sInit.EnableInEveryMode   :=TRUE;

(* Init ST03_422_B64_4 Zuführung ISK auf Übergabeposition Robo Palettierer (DigIn) *)
ST03_422_B64_4.sInit.InstName            :='ST03_421_B64_4';
ST03_422_B64_4.sInit.Description         :='Zuführung ISK auf Übergabeposition Robo Palettierer';
ST03_422_B64_4.sInit.BitInName           :='+8-421_B64.4';
ST03_422_B64_4.sInit.HomePosSignal       :=2; (* 0: Signal=Low, 1: Signal=High, 2: always  *)
ST03_422_B64_4.sInit.MaxTime             :=2000;
ST03_422_B64_4.sInit.EnableInEveryMode   :=TRUE;

(* Init ST03_422_Y64_5 Förderband  Zuführung Vereinzler AST/GST (Valve) *)
ST03_422_Y64_5.sInit.InstName            :='ST03_422_Y64_5';
ST03_422_Y64_5.sInit.BitName            :='+8-419_Y64.5';
ST03_422_Y64_5.sInit.Description         :='Förderband  Zuführung Vereinzler AST/GST';
ST03_422_Y64_5.sInit.HomePosDefine       :=HOME_ALWAYS;
ST03_422_Y64_5.sInit.InitDescription     :='GS einfahren';
ST03_422_Y64_5.sInit.WorkDescription     :='AS ausfahren';
ST03_422_Y64_5.sInit.DampBothTime        :=200;
ST03_422_Y64_5.sInit.KindOfValve         :='A';
ST03_422_Y64_5.sInit.MaxTime             :=2000;

(* Init ST03_422_Y64_6 Förderband  Stopper Vereinzler AST/GST (Valve) *)
ST03_422_Y64_6.sInit.InstName            :='ST03_422_Y64_6';
ST03_422_Y64_6.sInit.BitName            :='+8-419_Y64.6';
ST03_422_Y64_6.sInit.Description         :='Förderband  Stopper Vereinzler AST/GST';
ST03_422_Y64_6.sInit.HomePosDefine       :=HOME_ALWAYS;
ST03_422_Y64_6.sInit.InitDescription     :='GS ausfahren';
ST03_422_Y64_6.sInit.WorkDescription     :='AS einfahren';
ST03_422_Y64_6.sInit.DampBothTime        :=200;
ST03_422_Y64_6.sInit.KindOfValve         :='A';
ST03_422_Y64_6.sInit.MaxTime             :=2000;

(* Init ST03_422_Y64_7 Förderband  Stopper 1 Kamera AST/GST (Valve) *)
ST03_422_Y64_7.sInit.InstName            :='ST03_422_Y64_7';
ST03_422_Y64_7.sInit.BitName            :='+8-419_Y64.7';
ST03_422_Y64_7.sInit.Description         :='Förderband  Stopper Kamera AST/GST';
ST03_422_Y64_7.sInit.HomePosDefine       :=HOME_ALWAYS;
ST03_422_Y64_7.sInit.InitDescription     :='GS ausfahren';
ST03_422_Y64_7.sInit.WorkDescription     :='AS einfahren';
ST03_422_Y64_7.sInit.DampBothTime        :=200;
ST03_422_Y64_7.sInit.KindOfValve         :='A';
ST03_422_Y64_7.sInit.MaxTime             :=2000;

(* Init ST03_423_Y65_6 Förderband  Stopper 2 Kamera AST/GST (Valve) *)
ST03_423_Y65_6.sInit.InstName            :='ST03_423_Y65_6';
ST03_423_Y65_6.sInit.BitName            :='+8-423_Y65.6';
ST03_423_Y65_6.sInit.Description         :='Förderband  Stopper Kamera AST/GST';
ST03_423_Y65_6.sInit.HomePosDefine       :=HOME_ALWAYS;
ST03_423_Y65_6.sInit.InitDescription     :='GS ausfahren';
ST03_423_Y65_6.sInit.WorkDescription     :='AS einfahren';
ST03_423_Y65_6.sInit.DampBothTime        :=200;
ST03_423_Y65_6.sInit.KindOfValve         :='2G';
ST03_423_Y65_6.sInit.MaxTime             :=2000;

(* Init ST03_423_Y65_7 Förderband  Stopper 3 Kamera AST/GST (Valve) *)
ST03_423_Y65_7.sInit.InstName            :='ST03_423_Y65_7';
ST03_423_Y65_7.sInit.BitName            :='+8-423_Y65.7';
ST03_423_Y65_7.sInit.Description         :='Förderband  Stopper Kamera AST/GST';
ST03_423_Y65_7.sInit.HomePosDefine       :=HOME_ALWAYS;
ST03_423_Y65_7.sInit.InitDescription     :='GS ausfahren';
ST03_423_Y65_7.sInit.WorkDescription     :='AS einfahren';
ST03_423_Y65_7.sInit.DampBothTime        :=200;
ST03_423_Y65_7.sInit.KindOfValve         :='2G';
ST03_423_Y65_7.sInit.MaxTime             :=2000;

(* Init ST03_33F4 Steckdosen Tintenstrahldrucker (DigIn) *)
ST03_33F4.sInit.InstName            :='ST03_33_F4';
ST03_33F4.sInit.Description         :='SteckdosenTintenstrahldrucker';
ST03_33F4.sInit.BitInName           :='+33_F4';
ST03_33F4.sInit.HomePosSignal       :=2; (* 0: Signal=Low, 1: Signal=High, 2: always  *)
ST03_33F4.sInit.MaxTime             :=2000;
ST03_33F4.sInit.EnableInEveryMode   :=TRUE;

(* Init ST03_70U3_1 Bereit/ Im Druck Tintenstrahldrucker Frontseite (DigIn) *)
ST03_70U3_1.sInit.InstName            :='ST03_70U3_1';
ST03_70U3_1.sInit.Description         :='Bereit/ Im Druck Frontseite';
ST03_70U3_1.sInit.BitInName           :='+70U3_1';
ST03_70U3_1.sInit.HomePosSignal       :=2; (* 0: Signal=Low, 1: Signal=High, 2: always  *)
ST03_70U3_1.sInit.MaxTime             :=2000;
ST03_70U3_1.sInit.EnableInEveryMode   :=TRUE;

(* Init ST03_70U3_2 Tank voll Tintenstrahldrucker Frontseite (DigIn) *)
ST03_70U3_2.sInit.InstName            :='ST03_70U3_2';
ST03_70U3_2.sInit.Description         :='Tank voll Drucker Frontseite';
ST03_70U3_2.sInit.BitInName           :='+70U3_2';
ST03_70U3_2.sInit.HomePosSignal       :=2; (* 0: Signal=Low, 1: Signal=High, 2: always  *)
ST03_70U3_2.sInit.MaxTime             :=2000;
ST03_70U3_2.sInit.EnableInEveryMode   :=TRUE;

(* Init ST03_70U3_3 Fehler/Störung Tintenstrahldrucker Frontseite (DigIn) *)
ST03_70U3_3.sInit.InstName            :='ST03_70U3_3';
ST03_70U3_3.sInit.Description         :='Fehler Drucker Frontseite';
ST03_70U3_3.sInit.BitInName           :='+70U3_3';
ST03_70U3_3.sInit.HomePosSignal       :=2; (* 0: Signal=Low, 1: Signal=High, 2: always  *)
ST03_70U3_3.sInit.MaxTime             :=2000;
ST03_70U3_3.sInit.EnableInEveryMode   :=TRUE;

(* Init ST03_71U3_1 Bereit/ Im Druck Tintenstrahldrucker Rückseite (DigIn) *)
ST03_71U3_1.sInit.InstName            :='ST03_71U3_1';
ST03_71U3_1.sInit.Description         :='Bereit/ Im Druck  Rückseite';
ST03_71U3_1.sInit.BitInName           :='+71U3_1';
ST03_71U3_1.sInit.HomePosSignal       :=2; (* 0: Signal=Low, 1: Signal=High, 2: always  *)
ST03_71U3_1.sInit.MaxTime             :=2000;
ST03_71U3_1.sInit.EnableInEveryMode   :=TRUE;

(* Init ST03_71U3_2 Tank voll Tintenstrahldrucker Rückseite (DigIn) *)
ST03_71U3_2.sInit.InstName            :='ST03_71U3_2';
ST03_71U3_2.sInit.Description         :='Tank voll Drucker Rückseite';
ST03_71U3_2.sInit.BitInName           :='+71U3_2';
ST03_71U3_2.sInit.HomePosSignal       :=2; (* 0: Signal=Low, 1: Signal=High, 2: always  *)
ST03_71U3_2.sInit.MaxTime             :=2000;
ST03_71U3_2.sInit.EnableInEveryMode   :=TRUE;

(* Init ST03_71U3_3 Steckdosenleise (DigIn) *)
ST03_71U3_3.sInit.InstName            :='ST03_71U3_3';
ST03_71U3_3.sInit.Description         :='Fehler Drucker Rückseite';
ST03_71U3_3.sInit.BitInName           :='+71U3_3';
ST03_71U3_3.sInit.HomePosSignal       :=2; (* 0: Signal=Low, 1: Signal=High, 2: always  *)
ST03_71U3_3.sInit.MaxTime             :=2000;
ST03_71U3_3.sInit.EnableInEveryMode   :=TRUE;

(* Init ST03_PLAN_70V1_1 Start  Bedrucken Tintenstrahldrucker Frontseite (DigOutIn) *)
ST03_PLAN_70V1_1.sInit.InstName               :='ST03_PLAN_70V1_1';
ST03_PLAN_70V1_1.sInit.Description            :='Start  Drucker Frontseite';
ST03_PLAN_70V1_1.sInit.BitOutName             :='+PLAN_70V1_1';
ST03_PLAN_70V1_1.sInit.BitInName              :='';
ST03_PLAN_70V1_1.sInit.HomePosOutput          :=2; (* 0: Signal=Low, 1: Signal=High, 2: always  *)
ST03_PLAN_70V1_1.sInit.MaxTime                :=2000;
ST03_PLAN_70V1_1.sInit.EnableInEveryMode  :=TRUE;

(* Init ST03_PLAN_71V1_2 Start  Bedrucken Tintenstrahldrucker Rückseite (DigOutIn) *)
ST03_PLAN_71V1_2.sInit.InstName               :='ST03_PLAN_71V1_2';
ST03_PLAN_71V1_2.sInit.Description            :='Start  Drucker Rückseite';
ST03_PLAN_71V1_2.sInit.BitOutName             :='+PLAN_71V1_2';
ST03_PLAN_71V1_2.sInit.BitInName              :='';
ST03_PLAN_71V1_2.sInit.HomePosOutput          :=2; (* 0: Signal=Low, 1: Signal=High, 2: always  *)
ST03_PLAN_71V1_2.sInit.MaxTime                :=2000;
ST03_PLAN_71V1_2.sInit.EnableInEveryMode  :=TRUE;

(* Init ST03_Y01 Einschaltventil Hauptluft Tintenstrahldrucker (Valve) *)
ST03_Y01.sInit.InstName          :='ST03_Y01';
ST03_Y01.sInit.InstName          :='+Y01';
ST03_Y01.sInit.Description       :='Hauptluft Tintenstrahldrucker';
ST03_Y01.sInit.HomePosDefine     :=HOME_ALWAYS;
ST03_Y01.sInit.InitDescription   :='ON';
ST03_Y01.sInit.WorkDescription   :='OFF';
ST03_Y01.sInit.DampBothTime      :=0;
ST03_Y01.sInit.MaxTime           :=2000;
ST03_Y01.sInit.KindOfValve       :='A';

(* Init ST03_S18 ST02 Druckschalter Wartungseinheit Hauptluft Tintenstrahldrucker min.6 bar (DigIn) ST02_35_S31*)
ST03_S18.sInit.InstName            :='ST03_S18';
ST03_S18.sInit.Description         :='ST02 Druckschalter Wartungseinheit Hauptluft min.6 bar';
ST03_S18.sInit.BitInName           :='-ST03_S18';
ST03_S18.sInit.HomePosSignal       :=2; (* 0: Signal=Low, 1: Signal=High, 2: always  *)
ST03_S18.sInit.MaxTime             :=2000;
ST03_S18.sInit.EnableInEveryMode   :=TRUE;

(* Init ST03_H6 Signalsäule GR Bedruckung IO (DigOutIn) *)
ST03_H6.sInit.InstName               :='ST03_H6';
ST03_H6.sInit.Description            :='Signalsäule GR Bedruckung IO';
ST03_H6.sInit.BitOutName             :='-H6';
ST03_H6.sInit.BitInName              :='';
ST03_H6.sInit.HomePosOutput          :=2; (* 0: Signal=Low, 1: Signal=High, 2: always  *)
ST03_H6.sInit.MaxTime                :=2000;
ST03_H6.sInit.EnableInEveryMode   	 :=TRUE;

(* Init ST03_H7 Signalsäule RD Sammelstörung Bedruckung (DigOutIn) *)
ST03_H7.sInit.InstName               :='ST03_H7';
ST03_H7.sInit.Description            :='Signalsäule GR Bedruckung IO';
ST03_H7.sInit.BitOutName             :='-H7';
ST03_H7.sInit.BitInName              :='';
ST03_H7.sInit.HomePosOutput          :=2; (* 0: Signal=Low, 1: Signal=High, 2: always  *)
ST03_H7.sInit.MaxTime                :=2000;
ST03_H7.sInit.EnableInEveryMode   	 :=TRUE;
END_ACTION
ACTION Init_191pol:
(*Rüstsatz 191 pol ==================================================================================*)

(* Init ST03_541_B69_0 Zuführung  frei zum Ablegen ISK SP Maschine (DigIn) *)
ST03_541_B69_0.sInit.InstName            :='ST03_541_B69_0';
ST03_541_B69_0.sInit.Description         :='frei zum Ablegen ISK SP Maschine';
ST03_541_B69_0.sInit.BitInName           :='+8-541_B69.0';
ST03_541_B69_0.sInit.HomePosSignal       :=2; (* 0: Signal=Low, 1: Signal=High, 2: always  *)
ST03_541_B69_0.sInit.MaxTime             :=2000;
ST03_541_B69_0.sInit.EnableInEveryMode   :=TRUE;

(* Init ST03_541_B69_1 Zuführung Vereinzler eingefahren GST (ValveSensor) *)
ST03_541_B69_1.sInit.InstName		:='ST03_541_B69_1';
ST03_541_B69_1.sInit.BitName		:='+8_541_B69.1';
ST03_541_B69_1.sInit.Description	:=' Vereinzler eingefahren GST';
ST03_541_B69_1.sInit.SensorType	:=sValveSensorType_INIT;

(* Init ST03_541_B69_2 Zuführung Vereinzler ausgefahren AST (ValveSensor) *)
ST03_541_B69_2.sInit.InstName		:='ST03_541_B69_2';
ST03_541_B69_2.sInit.BitName		:='+8_541_B69.2';
ST03_541_B69_2.sInit.Description	:=' Vereinzler ausgefahren AST';
ST03_541_B69_2.sInit.SensorType	:=sValveSensorType_WORK;

(* Init ST03_541_B69_3 Zuführung Stopper eingefahren AST (ValveSensor) *)
ST03_541_B69_3.sInit.InstName		:='ST03_541_B69_3';
ST03_541_B69_3.sInit.BitName		:='+8_541_B69.3';
ST03_541_B69_3.sInit.Description	:='Stopper eingefahren AST';
ST03_541_B69_3.sInit.SensorType	:=sValveSensorType_WORK;

(* Init ST03_541_B69_4 Zuführung Stopper ausgefahren GST (ValveSensor) *)
ST03_541_B69_4.sInit.InstName		:='ST03_541_B69_4';
ST03_541_B69_4.sInit.BitName		:='+8_541_B69.4';
ST03_541_B69_4.sInit.Description	:='Stopper ausgefahren GST';
ST03_541_B69_4.sInit.SensorType	:=sValveSensorType_INIT;;

(* Init ST03_541_B69_6 ISK anwesend am Stopper (DigIn) *)
ST03_541_B69_6.sInit.InstName            :='ST03_541_B69_6';
ST03_541_B69_6.sInit.Description         :='ISK anwesend am Stopper';
ST03_541_B69_6.sInit.BitInName           :='+8-541_B69.6';
ST03_541_B69_6.sInit.HomePosSignal       :=2; (* 0: Signal=Low, 1: Signal=High, 2: always  *)
ST03_541_B69_6.sInit.MaxTime             :=2000;
ST03_541_B69_6.sInit.EnableInEveryMode   :=TRUE;

(* Init ST03_541_B69_7 ISK links Lageerkennung (DigIn) *)
ST03_541_B69_7.sInit.InstName            :='ST03_541_B69_7';
ST03_541_B69_7.sInit.Description         :='ISK links Lageerkennung.';
ST03_541_B69_7.sInit.BitInName           :='+8-541_B69.7';
ST03_541_B69_7.sInit.HomePosSignal       :=2; (* 0: Signal=Low, 1: Signal=High, 2: always  *)
ST03_541_B69_7.sInit.MaxTime             :=2000;
ST03_541_B69_7.sInit.EnableInEveryMode   :=TRUE;

(* Init ST03_542_B70_0 ISK rechts Lageerkennung (DigIn) *)
ST03_542_B70_0.sInit.InstName            :='ST03_542_B70_0';
ST03_542_B70_0.sInit.Description         :='ISK rechts Lageerkennung';
ST03_542_B70_0.sInit.BitInName           :='+8-542_B70.0';
ST03_542_B70_0.sInit.HomePosSignal       :=2; (* 0: Signal=Low, 1: Signal=High, 2: always  *)
ST03_542_B70_0.sInit.MaxTime             :=2000;
ST03_542_B70_0.sInit.EnableInEveryMode   :=TRUE;

(* Init ST03_542_Y70_1   Zuführung  Vereinzler AST/GST (Valve) *)
ST03_542_Y70_1.sInit.InstName            :='ST03_542_Y70_1';
ST03_542_Y70_1.sInit.BitName            :='+8-542_Y70.1';
ST03_542_Y70_1.sInit.Description         :=' Zuführung Vereinzler AST/GST';
ST03_542_Y70_1.sInit.HomePosDefine       :=HOME_ALWAYS;
ST03_542_Y70_1.sInit.InitDescription     :='GS einfahren';
ST03_542_Y70_1.sInit.WorkDescription     :='AS ausfahren';
ST03_542_Y70_1.sInit.DampBothTime        :=200;
ST03_542_Y70_1.sInit.KindOfValve         :='A';
ST03_542_Y70_1.sInit.MaxTime             :=2000;

(* Init ST03_542_Y70_2   Zuführung  Stopper AST/GST (Valve) *)
ST03_542_Y70_2.sInit.InstName            :='ST03_542_Y70_2';
ST03_542_Y70_2.sInit.BitName            :='+8-542_Y70.2';
ST03_542_Y70_2.sInit.Description         :=' Zuführung Stopper AST/GST';
ST03_542_Y70_2.sInit.HomePosDefine       :=HOME_ALWAYS;
ST03_542_Y70_2.sInit.InitDescription     :='GS ausfahren';
ST03_542_Y70_2.sInit.WorkDescription     :='AS einfahren';
ST03_542_Y70_2.sInit.DampBothTime        :=200;
ST03_542_Y70_2.sInit.KindOfValve         :='A';
ST03_542_Y70_2.sInit.MaxTime             :=2000;
END_ACTION
ACTION Init_206pol:
(*Rüstsatz 206pol*)
(* Init ST03_435_B67_0 Förderbandeinheit  Zuführung Vereinzler AST (ValveSensor) *)
ST03_435_B67_0.sInit.InstName            :='ST03_435_B67_0';
ST03_435_B67_0.sInit.BitName            :='+8_435_B67.0';
ST03_435_B67_0.sInit.Description         :='Förderbandeinheit  Zuführung Vereinzler AST';
ST03_435_B67_0.sInit.SensorType          :=sValveSensorType_INIT;

(* Init ST03_435_B67_1 Förderbandeinheit  Zuführung Vereinzler GST (ValveSensor) *)
ST03_435_B67_1.sInit.InstName            :='ST03_435_B67_1';
ST03_435_B67_1.sInit.BitName            :='+8_435_B67.1';
ST03_435_B67_1.sInit.Description         :='Förderbandeinheit  Zuführung Vereinzler GST';
ST03_435_B67_1.sInit.SensorType          :=sValveSensorType_WORK;

(* Init ST03_435_B67_2 Förderbandeinheit  Zuführung Stopper AST (ValveSensor) *)
ST03_435_B67_2.sInit.InstName            :='ST03_435_B67_2';
ST03_435_B67_2.sInit.BitName            :='+8_435_B67.2';
ST03_435_B67_2.sInit.Description         :='Förderband linke Zuführung Stopper AST';
ST03_435_B67_2.sInit.SensorType          :=sValveSensorType_INIT;

(* Init ST03_435_B67_3 Förderbandeinheit  Zuführung Stopper GST (ValveSensor) *)
ST03_435_B67_3.sInit.InstName            :='ST03_435_B67_3';
ST03_435_B67_3.sInit.BitName            :='+8_435_B67.3';
ST03_435_B67_3.sInit.Description         :='Förderband linke Zuführung Stopper GST';
ST03_435_B67_3.sInit.SensorType          :=sValveSensorType_WORK;

(* Init ST03_435_B67_4  Zuführung  frei zum Ablegen ISK SP Maschine Pos.1 (DigIn) *)
ST03_435_B67_4.sInit.InstName            :='ST03_435_B67_4';
ST03_435_B67_4.sInit.Description         :='Zuführung links frei zum Ablegen ISK SP Maschine Pos1';
ST03_435_B67_4.sInit.BitInName           :='+8-435_B67.4';
ST03_435_B67_4.sInit.HomePosSignal       :=2; (* 0: Signal=Low, 1: Signal=High, 2: always  *)
ST03_435_B67_4.sInit.MaxTime             :=2000;
ST03_435_B67_4.sInit.EnableInEveryMode   :=TRUE;

(* Init ST03_435_B67_7  ISK anwesend am Vereinzler (DigIn) *)
ST03_435_B67_7.sInit.InstName            :='ST03_435_B67_7';
ST03_435_B67_7.sInit.Description         :='ISK anwesend am Vereinzler';
ST03_435_B67_7.sInit.BitInName           :='+8-435_B67.7';
ST03_435_B67_7.sInit.HomePosSignal       :=2; (* 0: Signal=Low, 1: Signal=High, 2: always  *)
ST03_435_B67_7.sInit.MaxTime             :=2000;
ST03_435_B67_7.sInit.EnableInEveryMode   :=TRUE;

(* Init ST03_436_B68_1  Züführung  ISK Lageerkennung 1 (DigIn) *)
ST03_436_B68_1.sInit.InstName            :='ST03_436_B68_1';
ST03_436_B68_1.sInit.Description         :='Züführung  ISK Lageerkennung 1';
ST03_436_B68_1.sInit.BitInName           :='+8-436_B68.1';
ST03_436_B68_1.sInit.HomePosSignal       :=2; (* 0: Signal=Low, 1: Signal=High, 2: always  *)
ST03_436_B68_1.sInit.MaxTime             :=2000;
ST03_436_B68_1.sInit.EnableInEveryMode   :=TRUE;

(* Init ST03_436_B68_2  Züführung  ISK Lageerkennung 2 (DigIn) *)
ST03_436_B68_2.sInit.InstName            :='ST03_436_B68_2';
ST03_436_B68_2.sInit.Description         :='Züführung  ISK Lageerkennung 2';
ST03_436_B68_2.sInit.BitInName           :='+8-436_B68.2';
ST03_436_B68_2.sInit.HomePosSignal       :=2; (* 0: Signal=Low, 1: Signal=High, 2: always  *)
ST03_436_B68_2.sInit.MaxTime             :=2000;
ST03_436_B68_2.sInit.EnableInEveryMode   :=TRUE;

(* Init ST03_437_B68_4  ISK anwesend am Vereinzler (DigIn) *)
ST03_437_B68_4.sInit.InstName            :='ST03_437_B68_4';
ST03_437_B68_4.sInit.Description         :='Zuführung ISK auf Übergabeposition Robo Palettierer ';
ST03_437_B68_4.sInit.BitInName           :='+8-437_B68.4';
ST03_437_B68_4.sInit.HomePosSignal       :=2; (* 0: Signal=Low, 1: Signal=High, 2: always  *)
ST03_437_B68_4.sInit.MaxTime             :=2000;
ST03_437_B68_4.sInit.EnableInEveryMode   :=TRUE;

(* Init ST03_437_Y68_5 Förderband  Zuführung Vereinzler (Valve) *)
ST03_437_Y68_5.sInit.InstName            :='ST03_437_Y68_5';
ST03_437_Y68_5.sInit.BitName            :='+8-437_Y68.5';
ST03_437_Y68_5.sInit.Description         :='Förderband  Zuführung Vereinzler';
ST03_437_Y68_5.sInit.HomePosDefine       :=HOME_ALWAYS;
ST03_437_Y68_5.sInit.InitDescription     :='GS einfahren';
ST03_437_Y68_5.sInit.WorkDescription     :='AS ausfahren';
ST03_437_Y68_5.sInit.DampBothTime        :=200;
ST03_437_Y68_5.sInit.KindOfValve         :='A';
ST03_437_Y68_5.sInit.MaxTime             :=2000;

(* Init ST03_437_Y68_6 Förderband  Zuführung Stopper (Valve) *)
ST03_437_Y68_6.sInit.InstName            :='ST03_437_Y68_6';
ST03_437_Y68_6.sInit.BitName            :='+8-437_Y68.6';
ST03_437_Y68_6.sInit.Description         :='Förderband  Zuführung Stopper';
ST03_437_Y68_6.sInit.HomePosDefine       :=HOME_ALWAYS;
ST03_437_Y68_6.sInit.InitDescription     :='GS ausfahren';
ST03_437_Y68_6.sInit.WorkDescription     :='AS einfahren';
ST03_437_Y68_6.sInit.DampBothTime        :=200;
ST03_437_Y68_6.sInit.KindOfValve         :='A';
ST03_437_Y68_6.sInit.MaxTime             :=2000;
END_ACTION
ACTION Init_21pol:
(*Rüstsatz 21 pol ==================================================================================*)

(* Init ST03_536_B69_0 Zuführung  frei zum Ablegen ISK SP Maschine (DigIn) *)
ST03_536_B69_0.sInit.InstName            :='ST03_536_B69_0';
ST03_536_B69_0.sInit.Description         :='frei zum Ablegen ISK SP Maschine';
ST03_536_B69_0.sInit.BitInName           :='+8-536_B69.0';
ST03_536_B69_0.sInit.HomePosSignal       :=2; (* 0: Signal=Low, 1: Signal=High, 2: always  *)
ST03_536_B69_0.sInit.MaxTime             :=2000;
ST03_536_B69_0.sInit.EnableInEveryMode   :=TRUE;

(* Init ST03_536_B69_1 Zuführung Vereinzler eingefahren GST (ValveSensor) *)
ST03_536_B69_1.sInit.InstName		:='ST03_536_B69_1';
ST03_536_B69_1.sInit.BitName		:='+8_536_B69.1';
ST03_536_B69_1.sInit.Description	:=' Vereinzler eingefahren GST';
ST03_536_B69_1.sInit.SensorType	:=sValveSensorType_INIT;

(* Init ST03_536_B69_2 Zuführung Vereinzler ausgefahren AST (ValveSensor) *)
ST03_536_B69_2.sInit.InstName		:='ST03_536_B69_2';
ST03_536_B69_2.sInit.BitName		:='+8_536_B69.2';
ST03_536_B69_2.sInit.Description	:=' Vereinzler ausgefahren AST';
ST03_536_B69_2.sInit.SensorType	:=sValveSensorType_WORK;

(* Init ST03_536_B69_3 Zuführung Stopper eingefahren AST (ValveSensor) *)
ST03_536_B69_3.sInit.InstName		:='ST03_536_B69_3';
ST03_536_B69_3.sInit.BitName		:='+8_536_B69.3';
ST03_536_B69_3.sInit.Description	:='Stopper eingefahren AST';
ST03_536_B69_3.sInit.SensorType	:=sValveSensorType_WORK;

(* Init ST03_536_B69_4 Zuführung Stopper ausgefahren GST (ValveSensor) *)
ST03_536_B69_4.sInit.InstName		:='ST03_536_B69_4';
ST03_536_B69_4.sInit.BitName		:='+8_536_B69.4';
ST03_536_B69_4.sInit.Description	:='Stopper ausgefahren GST';
ST03_536_B69_4.sInit.SensorType	:=sValveSensorType_INIT;;

(* Init ST03_536_B69_6 ISK anwesend am Stopper (DigIn) *)
ST03_536_B69_6.sInit.InstName            :='ST03_536_B69_6';
ST03_536_B69_6.sInit.Description         :='ISK anwesend am Stopper';
ST03_536_B69_6.sInit.BitInName           :='+8-536_B69.6';
ST03_536_B69_6.sInit.HomePosSignal       :=2; (* 0: Signal=Low, 1: Signal=High, 2: always  *)
ST03_536_B69_6.sInit.MaxTime             :=2000;
ST03_536_B69_6.sInit.EnableInEveryMode   :=TRUE;

(* Init ST03_536_B69_7 ISK anwesend an Abholposition (DigIn) *)
ST03_536_B69_7.sInit.InstName            :='ST03_536_B69_7';
ST03_536_B69_7.sInit.Description         :='ISK anwesend an Abholpos.';
ST03_536_B69_7.sInit.BitInName           :='+8-536_B69.7';
ST03_536_B69_7.sInit.HomePosSignal       :=2; (* 0: Signal=Low, 1: Signal=High, 2: always  *)
ST03_536_B69_7.sInit.MaxTime             :=2000;
ST03_536_B69_7.sInit.EnableInEveryMode   :=TRUE;

(* Init ST03_537_B70_0 SK Lageerkennung (DigIn) *)
ST03_537_B70_0.sInit.InstName            :='ST03_537_B70_0';
ST03_537_B70_0.sInit.Description         :='ISK Lageerkennung';
ST03_537_B70_0.sInit.BitInName           :='+8-537_B70.0';
ST03_537_B70_0.sInit.HomePosSignal       :=2; (* 0: Signal=Low, 1: Signal=High, 2: always  *)
ST03_537_B70_0.sInit.MaxTime             :=2000;
ST03_537_B70_0.sInit.EnableInEveryMode   :=TRUE;

(* Init ST03_537_Y70_1   Zuführung  Vereinzler AST/GST (Valve) *)
ST03_537_Y70_1.sInit.InstName            :='ST03_537_Y70_1';
ST03_537_Y70_1.sInit.BitName            :='+8-537_Y70.1';
ST03_537_Y70_1.sInit.Description         :=' Zuführung Vereinzler AST/GST';
ST03_537_Y70_1.sInit.HomePosDefine       :=HOME_ALWAYS;
ST03_537_Y70_1.sInit.InitDescription     :='GS einfahren';
ST03_537_Y70_1.sInit.WorkDescription     :='AS ausfahren';
ST03_537_Y70_1.sInit.DampBothTime        :=200;
ST03_537_Y70_1.sInit.KindOfValve         :='A';
ST03_537_Y70_1.sInit.MaxTime             :=2000;

(* Init ST03_537_Y70_2   Zuführung  Stopper AST/GST (Valve) *)
ST03_537_Y70_2.sInit.InstName            :='ST03_537_Y70_2';
ST03_537_Y70_2.sInit.BitName            :='+8-537_Y70.2';
ST03_537_Y70_2.sInit.Description         :=' Zuführung Stopper AST/GST';
ST03_537_Y70_2.sInit.HomePosDefine       :=HOME_ALWAYS;
ST03_537_Y70_2.sInit.InitDescription     :='GS ausfahren';
ST03_537_Y70_2.sInit.WorkDescription     :='AS einfahren';
ST03_537_Y70_2.sInit.DampBothTime        :=200;
ST03_537_Y70_2.sInit.KindOfValve         :='A';
ST03_537_Y70_2.sInit.MaxTime             :=2000;
END_ACTION
ACTION Init_268pol_102pol_neu:
(*Rüstsatz 268 pol ==================================================================================*)

(* Init ST03_556_B69_0 Zuführung  frei zum Ablegen ISK SP Maschine (DigIn) *)
ST03_556_B69_0.sInit.InstName            :='ST03_556_B69_0';
ST03_556_B69_0.sInit.Description         :='frei zum Ablegen ISK SP Maschine';
ST03_556_B69_0.sInit.BitInName           :='+8_556_B69.0';
ST03_556_B69_0.sInit.HomePosSignal       :=2; (* 0: Signal=Low, 1: Signal=High, 2: always  *)
ST03_556_B69_0.sInit.MaxTime             :=2000;
ST03_556_B69_0.sInit.EnableInEveryMode   :=TRUE;

(* Init ST03_556_B69_1 Zuführung Vereinzler eingefahren GST (ValveSensor) *)
ST03_556_B69_1.sInit.InstName		:='ST03_556_B69_1';
ST03_556_B69_1.sInit.BitName		:='+8_556_B69.1';
ST03_556_B69_1.sInit.Description	:=' Vereinzler eingefahren GST';
ST03_556_B69_1.sInit.SensorType	:=sValveSensorType_INIT;

(* Init ST03_556_B69_2 Zuführung Vereinzler ausgefahren AST (ValveSensor) *)
ST03_556_B69_2.sInit.InstName		:='ST03_556_B69_2';
ST03_556_B69_2.sInit.BitName		:='+8_556_B69.2';
ST03_556_B69_2.sInit.Description	:=' Vereinzler ausgefahren AST';
ST03_556_B69_2.sInit.SensorType	:=sValveSensorType_WORK;

(* Init ST03_556_B69_3 Zuführung Stopper eingefahren AST (ValveSensor) *)
ST03_556_B69_3.sInit.InstName		:='ST03_556_B69_3';
ST03_556_B69_3.sInit.BitName		:='+8_556_B69.3';
ST03_556_B69_3.sInit.Description	:='Stopper eingefahren AST';
ST03_556_B69_3.sInit.SensorType	:=sValveSensorType_WORK;

(* Init ST03_556_B69_4 Zuführung Stopper ausgefahren GST (ValveSensor) *)
ST03_556_B69_4.sInit.InstName		:='ST03_556_B69_4';
ST03_556_B69_4.sInit.BitName		:='+8_556_B69.4';
ST03_556_B69_4.sInit.Description	:='Stopper ausgefahren GST';
ST03_556_B69_4.sInit.SensorType	:=sValveSensorType_INIT;;

(* Init ST03_556_B69_5  Führungsschiene Überwachung Staustrecke (DigIn) *)
ST03_556_B69_5.sInit.InstName            :='ST03_556_B69_5';
ST03_556_B69_5.sInit.Description         :='Führungsschiene Überwachung Staustrecke';
ST03_556_B69_5.sInit.BitInName           :='+8_556_B69.5';
ST03_556_B69_5.sInit.HomePosSignal       :=2; (* 0: Signal=Low, 1: Signal=High, 2: always  *)
ST03_556_B69_5.sInit.MaxTime             :=2000;
ST03_556_B69_5.sInit.EnableInEveryMode   :=TRUE;

(* Init ST03_556_B69_6 ISK anwesend am Stopper (DigIn) *)
ST03_556_B69_6.sInit.InstName            :='ST03_556_B69_6';
ST03_556_B69_6.sInit.Description         :='ISK anwesend am Stopper';
ST03_556_B69_6.sInit.BitInName           :='+8_556_B69.6';
ST03_556_B69_6.sInit.HomePosSignal       :=2; (* 0: Signal=Low, 1: Signal=High, 2: always  *)
ST03_556_B69_6.sInit.MaxTime             :=2000;
ST03_556_B69_6.sInit.EnableInEveryMode   :=TRUE;

(* Init ST03_556_B69_7 ISK  auf Übergabeposition  (DigIn) *)
ST03_556_B69_7.sInit.InstName            :='ST03_556_B69_7';
ST03_556_B69_7.sInit.Description         :='ISK  auf Übergabeposition .';
ST03_556_B69_7.sInit.BitInName           :='+8_556_B69.7';
ST03_556_B69_7.sInit.HomePosSignal       :=2; (* 0: Signal=Low, 1: Signal=High, 2: always  *)
ST03_556_B69_7.sInit.MaxTime             :=2000;
ST03_556_B69_7.sInit.EnableInEveryMode   :=TRUE;

(* Init ST03_557_Y70_1   Zuführung  Vereinzler AST/GST (Valve) *)
ST03_557_Y70_1.sInit.InstName            :='ST03_557_Y70_1';
ST03_557_Y70_1.sInit.BitName            :='+8_557_Y70.1';
ST03_557_Y70_1.sInit.Description         :=' Zuführung Vereinzler AST/GST';
ST03_557_Y70_1.sInit.HomePosDefine       :=HOME_ALWAYS;
ST03_557_Y70_1.sInit.InitDescription     :='GS einfahren';
ST03_557_Y70_1.sInit.WorkDescription     :='AS ausfahren';
ST03_557_Y70_1.sInit.DampBothTime        :=200;
ST03_557_Y70_1.sInit.KindOfValve         :='A';
ST03_557_Y70_1.sInit.MaxTime             :=2000;

(* Init ST03_557_Y70_2   Zuführung  Stopper AST/GST (Valve) *)
ST03_557_Y70_2.sInit.InstName            :='ST03_557_Y70_2';
ST03_557_Y70_2.sInit.BitName            :='+8_557_Y70.2';
ST03_557_Y70_2.sInit.Description         :=' Zuführung Stopper AST/GST';
ST03_557_Y70_2.sInit.HomePosDefine       :=HOME_ALWAYS;
ST03_557_Y70_2.sInit.InitDescription     :='GS ausfahren';
ST03_557_Y70_2.sInit.WorkDescription     :='AS einfahren';
ST03_557_Y70_2.sInit.DampBothTime        :=200;
ST03_557_Y70_2.sInit.KindOfValve         :='A';
ST03_557_Y70_2.sInit.MaxTime             :=2000;
END_ACTION
ACTION Init_268polRP:
(*Rüstsatz 268 pol Rasterplatte==================================================================================*)

(* Init ST03_562_B69_0 Zuführung 1 frei zum Schwenken (DigIn) *)
ST03_562_B69_0.sInit.InstName            :='ST03_562_B69_0';
ST03_562_B69_0.sInit.Description         :='Zuführung 1 frei zum Schwenken';
ST03_562_B69_0.sInit.BitInName           :='+8-562_B71.7';
ST03_562_B69_0.sInit.HomePosSignal       :=2; (* 0: Signal=Low, 1: Signal=High, 2: always  *)
ST03_562_B69_0.sInit.MaxTime             :=2000;
ST03_562_B69_0.sInit.EnableInEveryMode   :=TRUE;

(* Init ST03_562_B69_1 Zuführung 1 Vereinzler GST (ValveSensor) *)
ST03_562_B69_1.sInit.InstName		:='ST03_562_B69_1';
ST03_562_B69_1.sInit.BitName		:='+8_562_B69.1';
ST03_562_B69_1.sInit.Description	:='Zuführung 1 Vereinzler GST';
ST03_562_B69_1.sInit.SensorType	:=sValveSensorType_INIT;

(* Init ST03_562_B69_2 Zuführung 1 Vereinzler AST (ValveSensor) *)
ST03_562_B69_2.sInit.InstName		:='ST03_562_B69_2';
ST03_562_B69_2.sInit.BitName		:='+8_562_B69.2';
ST03_562_B69_2.sInit.Description	:='Zuführung 1 Vereinzler AST';
ST03_562_B69_2.sInit.SensorType	:=sValveSensorType_WORK;

(* Init ST03_562_B69_3 Zuführung 1 Stopper AST (ValveSensor) *)
ST03_562_B69_3.sInit.InstName		:='ST03_562_B69_3';
ST03_562_B69_3.sInit.BitName		:='+8_562_B69.3';
ST03_562_B69_3.sInit.Description	:='Zuführung 1 Stopper AST';
ST03_562_B69_3.sInit.SensorType	:=sValveSensorType_WORK;

(* Init ST03_562_B69_4 Zuführung 1 Stopper GST (ValveSensor) *)
ST03_562_B69_4.sInit.InstName		:='ST03_562_B69_4';
ST03_562_B69_4.sInit.BitName		:='+8_562_B69.4';
ST03_562_B69_4.sInit.Description	:='Zuführung 1 Stopper GST';
ST03_562_B69_4.sInit.SensorType	:=sValveSensorType_INIT;

(* Init ST03_562_B69_6 Zuführung 1 ISK anwesend am Stopper (DigIn) *)
ST03_562_B69_6.sInit.InstName            :='ST03_562_B69_6';
ST03_562_B69_6.sInit.Description         :='Zuführung 1 ISK anwesend am Stopper';
ST03_562_B69_6.sInit.BitInName           :='+8-562_B69.6';
ST03_562_B69_6.sInit.HomePosSignal       :=2; (* 0: Signal=Low, 1: Signal=High, 2: always  *)
ST03_562_B69_6.sInit.MaxTime             :=2000;
ST03_562_B69_6.sInit.EnableInEveryMode   :=TRUE;

(* Init ST03_562_B67_7 Zuführung 1 ISK auf Übergabepos. Robi (DigIn) *)
ST03_562_B67_7.sInit.InstName            :='ST03_562_B67_7';
ST03_562_B67_7.sInit.Description         :='Zuführung 1 ISK auf Übergabepos. Robi';
ST03_562_B67_7.sInit.BitInName           :='+8-562_B69.7';
ST03_562_B67_7.sInit.HomePosSignal       :=2; (* 0: Signal=Low, 1: Signal=High, 2: always  *)
ST03_562_B67_7.sInit.MaxTime             :=2000;
ST03_562_B67_7.sInit.EnableInEveryMode   :=TRUE;

(* Init ST03_563_B70_0 Zuführung 2 frei zum Schwenken (DigIn) *)
ST03_563_B70_0.sInit.InstName            :='ST03_563_B70_0';
ST03_563_B70_0.sInit.Description         :='Zuführung 2 frei zum Schwenken';
ST03_563_B70_0.sInit.BitInName           :='+8-563_B71.7';
ST03_563_B70_0.sInit.HomePosSignal       :=2; (* 0: Signal=Low, 1: Signal=High, 2: always  *)
ST03_563_B70_0.sInit.MaxTime             :=2000;
ST03_563_B70_0.sInit.EnableInEveryMode   :=TRUE;

(* Init ST03_563_B70_1 Zuführung 2 Vereinzler GAST (ValveSensor) *)
ST03_563_B70_1.sInit.InstName		:='ST03_563_B70_1';
ST03_563_B70_1.sInit.BitName		:='+8_563_B70.1';
ST03_563_B70_1.sInit.Description	:='Zuführung 2 Vereinzler GST';
ST03_563_B70_1.sInit.SensorType	:=sValveSensorType_INIT;

(* Init ST03_563_B70_2 Zuführung 2 Vereinzler AST (ValveSensor) *)
ST03_563_B70_2.sInit.InstName		:='ST03_563_B70_2';
ST03_563_B70_2.sInit.BitName		:='+8_563_B70.2';
ST03_563_B70_2.sInit.Description	:='Zuführung 2 Vereinzler AST';
ST03_563_B70_2.sInit.SensorType	:=sValveSensorType_WORK;

(* Init ST03_563_B70_3 Zuführung 2 Stopper AST (ValveSensor) *)
ST03_563_B70_3.sInit.InstName		:='ST03_563_B70_3';
ST03_563_B70_3.sInit.BitName		:='+8_563_B70.3';
ST03_563_B70_3.sInit.Description	:='Zuführung 2 Stopper AST';
ST03_563_B70_3.sInit.SensorType	:=sValveSensorType_WORK;

(* Init ST03_563_B70_4 Zuführung 2 Stopper GST (ValveSensor) *)
ST03_563_B70_4.sInit.InstName		:='ST03_563_B70_4';
ST03_563_B70_4.sInit.BitName		:='+8_563_B70.4';
ST03_563_B70_4.sInit.Description	:='Zuführung 2 Stopper GST';
ST03_563_B70_4.sInit.SensorType	:=sValveSensorType_INIT;

(* Init ST03_563_B70_6 Zuführung 2 ISK anwesend am Stopper (DigIn) *)
ST03_563_B70_6.sInit.InstName            :='ST03_563_B70_6';
ST03_563_B70_6.sInit.Description         :='Zuführung 2 ISK anwesend am Stopper';
ST03_563_B70_6.sInit.BitInName           :='+8-563_B70.6';
ST03_563_B70_6.sInit.HomePosSignal       :=2; (* 0: Signal=Low, 1: Signal=High, 2: always  *)
ST03_563_B70_6.sInit.MaxTime             :=2000;
ST03_563_B70_6.sInit.EnableInEveryMode   :=TRUE;

(* Init ST03_563_B70_7 Zuführung 2 ISK auf Übergabepos. Robi (DigIn) *)
ST03_563_B70_7.sInit.InstName            :='ST03_563_B70_7';
ST03_563_B70_7.sInit.Description         :='Zuführung 2 ISK auf Übergabepos. Robi';
ST03_563_B70_7.sInit.BitInName           :='+8-563_B70.7';
ST03_563_B70_7.sInit.HomePosSignal       :=2; (* 0: Signal=Low, 1: Signal=High, 2: always  *)
ST03_563_B70_7.sInit.MaxTime             :=2000;
ST03_563_B70_7.sInit.EnableInEveryMode   :=TRUE;

(* Init ST03_564_Y71_0  Zuführung 1 Vereinzler   AST/GST (Valve) *)
ST03_564_Y71_0.sInit.InstName            :='ST03_564_Y71_0';
ST03_564_Y71_0.sInit.BitName            :='+8-564_Y71.0';
ST03_564_Y71_0.sInit.Description         :='Zuführung 1 Vereinzler AST/GST';
ST03_564_Y71_0.sInit.HomePosDefine       :=HOME_ALWAYS;
ST03_564_Y71_0.sInit.InitDescription     :='GS einfahren';
ST03_564_Y71_0.sInit.WorkDescription     :='AS ausfahren';
ST03_564_Y71_0.sInit.DampBothTime        :=200;
ST03_564_Y71_0.sInit.KindOfValve         :='A';
ST03_564_Y71_0.sInit.MaxTime             :=2000;

(* Init ST03_564_Y71_1  Zuführung 1 Stopper   AST/GST (Valve) *)
ST03_564_Y71_1.sInit.InstName            :='ST03_564_Y71_1';
ST03_564_Y71_1.sInit.BitName            :='+8-564_Y71.1';
ST03_564_Y71_1.sInit.Description         :='Zuführung 1 Stopper AST/GST';
ST03_564_Y71_1.sInit.HomePosDefine       :=HOME_ALWAYS;
ST03_564_Y71_1.sInit.InitDescription     :='GS ausfahren';
ST03_564_Y71_1.sInit.WorkDescription     :='AS einfahren';
ST03_564_Y71_1.sInit.DampBothTime        :=200;
ST03_564_Y71_1.sInit.KindOfValve         :='A';
ST03_564_Y71_1.sInit.MaxTime             :=2000;

(* Init ST03_564_Y71_2  Zuführung 2 Vereinzler   AST/GST (Valve) *)
ST03_564_Y71_2.sInit.InstName            :='ST03_564_Y71_2';
ST03_564_Y71_2.sInit.BitName            :='+8-564_Y71.2';
ST03_564_Y71_2.sInit.Description         :='Zuführung 2 Vereinzler AST/GST';
ST03_564_Y71_2.sInit.HomePosDefine       :=HOME_ALWAYS;
ST03_564_Y71_2.sInit.InitDescription     :='GS einfahren';
ST03_564_Y71_2.sInit.WorkDescription     :='AS ausfahren';
ST03_564_Y71_2.sInit.DampBothTime        :=200;
ST03_564_Y71_2.sInit.KindOfValve         :='A';
ST03_564_Y71_2.sInit.MaxTime             :=2000;

(* Init ST03_564_Y71_3  Zuführung 2 Stopper   AST/GST (Valve) *)
ST03_564_Y71_3.sInit.InstName            :='ST03_564_Y71_3';
ST03_564_Y71_3.sInit.BitName            :='+8-564_Y71.3';
ST03_564_Y71_3.sInit.Description         :='Zuführung 2 Stopper AST/GST';
ST03_564_Y71_3.sInit.HomePosDefine       :=HOME_ALWAYS;
ST03_564_Y71_3.sInit.InitDescription     :='GS ausfahren';
ST03_564_Y71_3.sInit.WorkDescription     :='AS einfahren';
ST03_564_Y71_3.sInit.DampBothTime        :=200;
ST03_564_Y71_3.sInit.KindOfValve         :='A';
ST03_564_Y71_3.sInit.MaxTime             :=2000;

(* Init ST03_564_Y71_4   ISK Klemmer AST/GST (Valve) *)
ST03_564_Y71_4.sInit.InstName            :='ST03_564_Y71_4';
ST03_564_Y71_4.sInit.BitName            :='+8-564_Y71.4';
ST03_564_Y71_4.sInit.Description         :=' ISK Klemmer AST/GST';
ST03_564_Y71_4.sInit.HomePosDefine       :=HOME_ALWAYS;
ST03_564_Y71_4.sInit.InitDescription     :='GS auf';
ST03_564_Y71_4.sInit.WorkDescription     :='AS zu';
ST03_564_Y71_4.sInit.DampBothTime        :=200;
ST03_564_Y71_4.sInit.KindOfValve         :='A';
ST03_564_Y71_4.sInit.MaxTime             :=2000;

(* Init ST03_564_Y71_5  Rinne schwenkern  AST/GST (Valve) *)
ST03_564_Y71_5.sInit.InstName            :='ST03_564_Y71_5';
ST03_564_Y71_5.sInit.BitName            :='+8-564_Y71.5';
ST03_564_Y71_5.sInit.Description         :=' Rinne schwenkern AST/GST';
ST03_564_Y71_5.sInit.HomePosDefine       :=HOME_ALWAYS;
ST03_564_Y71_5.sInit.InitDescription     :='GS 0 Grad';
ST03_564_Y71_5.sInit.WorkDescription     :='AS 180 Grad';
ST03_564_Y71_5.sInit.DampBothTime        :=200;
ST03_564_Y71_5.sInit.KindOfValve         :='A';
ST03_564_Y71_5.sInit.MaxTime             :=4000;

(* Init ST03_565_B72_0  ISK 1 in Klemme (DigIn) *)
ST03_565_B72_0.sInit.InstName            :='ST03_565_B72_0';
ST03_565_B72_0.sInit.Description         :=' ISK 1 in Klemme';
ST03_565_B72_0.sInit.BitInName           :='+8-565_B72.0';
ST03_565_B72_0.sInit.HomePosSignal       :=2; (* 0: Signal=Low, 1: Signal=High, 2: always  *)
ST03_565_B72_0.sInit.MaxTime             :=2000;
ST03_565_B72_0.sInit.EnableInEveryMode   :=TRUE;

(* Init ST03_565_B72_1  ISK 2 in Klemme (DigIn) *)
ST03_565_B72_1.sInit.InstName            :='ST03_565_B72_1';
ST03_565_B72_1.sInit.Description         :=' ISK 2 in Klemme';
ST03_565_B72_1.sInit.BitInName           :='+8-565_B72.1';
ST03_565_B72_1.sInit.HomePosSignal       :=2; (* 0: Signal=Low, 1: Signal=High, 2: always  *)
ST03_565_B72_1.sInit.MaxTime             :=2000;
ST03_565_B72_1.sInit.EnableInEveryMode   :=TRUE;

(* Init ST03_565_B72_2 'ISK Klemmer 1 offen GST (ValveSensor) *)
ST03_565_B72_2.sInit.InstName		:='ST03_565_B72_2';
ST03_565_B72_2.sInit.BitName		:='+8_565_B72.2';
ST03_565_B72_2.sInit.Description	:='ISK Klemmer 1 offen GST';
ST03_565_B72_2.sInit.SensorType	:=sValveSensorType_INIT;

(* Init ST03_565_B72_3 'ISK Klemmer 1 zu AST (ValveSensor) *)
ST03_565_B72_3.sInit.InstName		:='ST03_565_B72_3';
ST03_565_B72_3.sInit.BitName		:='+8_565_B72.3';
ST03_565_B72_3.sInit.Description	:='ISK Klemmer 1 zu AST';
ST03_565_B72_3.sInit.SensorType	:=sValveSensorType_WORK;

(* Init ST03_565_B72_4 'ISK Klemmer 2 offen GST (ValveSensor) *)
ST03_565_B72_4.sInit.InstName		:='ST03_565_B72_4';
ST03_565_B72_4.sInit.BitName		:='+8_565_B72.4';
ST03_565_B72_4.sInit.Description	:='ISK Klemmer 2 offen GST';
ST03_565_B72_4.sInit.SensorType	:=sValveSensorType_INIT;

(* Init ST03_565_B72_5 'ISK Klemmer 2 zu AST (ValveSensor) *)
ST03_565_B72_5.sInit.InstName		:='ST03_565_B72_5';
ST03_565_B72_5.sInit.BitName		:='+8_565_B72.5';
ST03_565_B72_5.sInit.Description	:='ISK Klemmer 2 zu AST';
ST03_565_B72_5.sInit.SensorType	:=sValveSensorType_WORK;

(* Init ST03_565_B72_6 Rinne schwenkern 0° AST (ValveSensor) *)
ST03_565_B72_6.sInit.InstName		:='ST03_565_B72_6';
ST03_565_B72_6.sInit.BitName		:='+8_565_B72.6';
ST03_565_B72_6.sInit.Description	:='Rinne schwenkern 0° AST';
ST03_565_B72_6.sInit.SensorType	:=sValveSensorType_WORK;

(* Init ST03_565_B72_7 Rinne schwenkern 180° GST (ValveSensor) *)
ST03_565_B72_7.sInit.InstName		:='ST03_565_B72_7';
ST03_565_B72_7.sInit.BitName		:='+8_565_B72.7';
ST03_565_B72_7.sInit.Description	:='Rinne schwenkern 180° GST';
ST03_565_B72_7.sInit.SensorType	:=sValveSensorType_INIT;
END_ACTION
ACTION Init_33pol:
(*Rüstsatz 33 pol ==================================================================================*)

(* Init ST03_556_B69_0 Zuführung Pos 1 frei zum Ablegen ISK SP Maschine (DigIn) *)
ST03_571_B69_0.sInit.InstName            :='ST03_571_B69_0';
ST03_571_B69_0.sInit.Description         :='Pos 1 frei zum Ablegen ISK SP Maschine';
ST03_571_B69_0.sInit.BitInName           :='+8_571_B69.0';
ST03_571_B69_0.sInit.HomePosSignal       :=2; (* 0: Signal=Low, 1: Signal=High, 2: always  *)
ST03_571_B69_0.sInit.MaxTime             :=2000;
ST03_571_B69_0.sInit.EnableInEveryMode   :=TRUE;

(* Init ST03_556_B69_1 Zuführung Pos 2 frei zum Ablegen ISK SP Maschine (DigIn) *)
ST03_571_B69_1.sInit.InstName            :='ST03_571_B69_1';
ST03_571_B69_1.sInit.Description         :='Pos 2 frei zum Ablegen ISK SP Maschine';
ST03_571_B69_1.sInit.BitInName           :='+8_571_B69.0';
ST03_571_B69_1.sInit.HomePosSignal       :=2; (* 0: Signal=Low, 1: Signal=High, 2: always  *)
ST03_571_B69_1.sInit.MaxTime             :=2000;
ST03_571_B69_1.sInit.EnableInEveryMode   :=TRUE;

(* Init ST03_571_B69_2 Zuführung Vereinzler eingefahren GST (ValveSensor) *)
ST03_571_B69_2.sInit.InstName		:='ST03_571_B69_2';
ST03_571_B69_2.sInit.BitName		:='+8_571_B69.2';
ST03_571_B69_2.sInit.Description	:=' Vereinzler eingefahren GST';
ST03_571_B69_2.sInit.SensorType	:=sValveSensorType_INIT;

(* Init ST03_571_B69_3 Zuführung Vereinzler ausgefahren AST (ValveSensor) *)
ST03_571_B69_3.sInit.InstName		:='ST03_571_B69_3';
ST03_571_B69_3.sInit.BitName		:='+8_571_B69.3';
ST03_571_B69_3.sInit.Description	:=' Vereinzler ausgefahren AST';
ST03_571_B69_3.sInit.SensorType	:=sValveSensorType_WORK;

(* Init ST03_571_B69_4 Zuführung Stopper eingefahren AST (ValveSensor) *)
ST03_571_B69_4.sInit.InstName		:='ST03_571_B69_4';
ST03_571_B69_4.sInit.BitName		:='+8_571_B69.4';
ST03_571_B69_4.sInit.Description	:='Stopper eingefahren AST';
ST03_571_B69_4.sInit.SensorType	:=sValveSensorType_WORK;

(* Init ST03_571_B69_5 Zuführung Stopper ausgefahren GST (ValveSensor) *)
ST03_571_B69_5.sInit.InstName		:='ST03_571_B69_5';
ST03_571_B69_5.sInit.BitName		:='+8_571_B69.5';
ST03_571_B69_5.sInit.Description	:='Stopper ausgefahren GST';
ST03_571_B69_5.sInit.SensorType	:=sValveSensorType_INIT;;

(* Init ST03_571_B69_6 ISK anwesend am Stopper (DigIn) *)
ST03_571_B69_6.sInit.InstName            :='ST03_571_B69_6';
ST03_571_B69_6.sInit.Description         :='ISK anwesend am Stopper';
ST03_571_B69_6.sInit.BitInName           :='+8_571_B69.6';
ST03_571_B69_6.sInit.HomePosSignal       :=2; (* 0: Signal=Low, 1: Signal=High, 2: always  *)
ST03_571_B69_6.sInit.MaxTime             :=2000;
ST03_571_B69_6.sInit.EnableInEveryMode   :=TRUE;

(* Init ST03_571_B69_7 ISK rechts Lageerkennung (DigIn) *)
ST03_571_B69_7.sInit.InstName            :='ST03_571_B69_7';
ST03_571_B69_7.sInit.Description         :='ISK rechts Lageerkennung.';
ST03_571_B69_7.sInit.BitInName           :='+8_571_B69.7';
ST03_571_B69_7.sInit.HomePosSignal       :=2; (* 0: Signal=Low, 1: Signal=High, 2: always  *)
ST03_571_B69_7.sInit.MaxTime             :=2000;
ST03_571_B69_7.sInit.EnableInEveryMode   :=TRUE;

(* Init ST03_572_Y70_0   Zuführung  Vereinzler AST/GST (Valve) *)
ST03_572_Y70_0.sInit.InstName            :='ST03_572_Y70_0';
ST03_572_Y70_0.sInit.BitName            :='+8_572_Y70.0';
ST03_572_Y70_0.sInit.Description         :='Zuführung Vereinzler AST/GST';
ST03_572_Y70_0.sInit.HomePosDefine       :=HOME_ALWAYS;
ST03_572_Y70_0.sInit.InitDescription     :='GS einfahren';
ST03_572_Y70_0.sInit.WorkDescription     :='AS ausfahren';
ST03_572_Y70_0.sInit.DampBothTime        :=200;
ST03_572_Y70_0.sInit.KindOfValve         :='A';
ST03_572_Y70_0.sInit.MaxTime             :=2000;

(* Init ST03_572_Y70_1   Zuführung  Stopper AST/GST (Valve) *)
ST03_572_Y70_1.sInit.InstName            :='ST03_572_Y70_1';
ST03_572_Y70_1.sInit.BitName            :='+8_572_Y70.1';
ST03_572_Y70_1.sInit.Description         :='Zuführung Stopper AST/GST';
ST03_572_Y70_1.sInit.HomePosDefine       :=HOME_ALWAYS;
ST03_572_Y70_1.sInit.InitDescription     :='GS ausfahren';
ST03_572_Y70_1.sInit.WorkDescription     :='AS einfahren';
ST03_572_Y70_1.sInit.DampBothTime        :=200;
ST03_572_Y70_1.sInit.KindOfValve         :='A';
ST03_572_Y70_1.sInit.MaxTime             :=2000;
END_ACTION
ACTION Init_46pol:
(*========================= Rüstsatz 46 polig===============================*)

(* Init ST03_461_B69_0 Förderbandeinheit  Zuführung Vereinzler AST (ValveSensor) *)
ST03_461_B69_0.sInit.InstName            :='ST03_461_B69_0';
ST03_461_B69_0.sInit.BitName            :='+8_461_B69.0';
ST03_461_B69_0.sInit.Description         :='Förderbandeinheit  Zuführung Vereinzler AST';
ST03_461_B69_0.sInit.SensorType          :=sValveSensorType_INIT;

(* Init ST03_461_B69_1 Förderbandeinheit  Zuführung Vereinzler GST (ValveSensor) *)
ST03_461_B69_1.sInit.InstName            :='ST03_461_B69_1';
ST03_461_B69_1.sInit.BitName            :='+8_461_B69.1';
ST03_461_B69_1.sInit.Description         :='Förderbandeinheit  Zuführung Vereinzler GST';
ST03_461_B69_1.sInit.SensorType          :=sValveSensorType_WORK;

(* Init ST03_461_B69_2 Förderbandeinheit  Zuführung Stopper AST (ValveSensor) *)
ST03_461_B69_2.sInit.InstName            :='ST03_461_B69_2';
ST03_461_B69_2.sInit.BitName            :='+8_461_B69.2';
ST03_461_B69_2.sInit.Description         :='Förderband linke Zuführung Stopper AST';
ST03_461_B69_2.sInit.SensorType          :=sValveSensorType_INIT;

(* Init ST03_461_B69_3 Förderbandeinheit  Zuführung Stopper GST (ValveSensor) *)
ST03_461_B69_3.sInit.InstName            :='ST03_461_B69_3';
ST03_461_B69_3.sInit.BitName            :='+8_461_B69.3';
ST03_461_B69_3.sInit.Description         :='Förderband linke Zuführung Stopper GST';
ST03_461_B69_3.sInit.SensorType          :=sValveSensorType_WORK;

(* Init ST03_461_B69_4  Zuführung  frei zum Ablegen ISK SP Maschine Pos.1 (DigIn) *)
ST03_461_B69_4.sInit.InstName            :='ST03_461_B69_4';
ST03_461_B69_4.sInit.Description         :='Zuführung links frei zum Ablegen ISK SP Maschine Pos1';
ST03_461_B69_4.sInit.BitInName           :='+8-461_B69.4';
ST03_461_B69_4.sInit.HomePosSignal       :=2; (* 0: Signal=Low, 1: Signal=High, 2: always  *)
ST03_461_B69_4.sInit.MaxTime             :=2000;
ST03_461_B69_4.sInit.EnableInEveryMode   :=TRUE;

(* Init ST03_461_B69_5 Förderbandeinheit  Zuführung Stopper GST (ValveSensor) *)
ST03_461_B69_5.sInit.InstName            :='ST03_461_B69_5';
ST03_461_B69_5.sInit.BitName            :='+8_461_B69.5';
ST03_461_B69_5.sInit.Description         :='Förderband  Vereinzelner Wender AST';
ST03_461_B69_5.sInit.SensorType          :=sValveSensorType_INIT;

(* Init ST03_461_B69_6 Förderbandeinheit  Zuführung Stopper GST (ValveSensor) *)
ST03_461_B69_6.sInit.InstName            :='ST03_461_B69_6';
ST03_461_B69_6.sInit.BitName            :='+8_461_B69.6';
ST03_461_B69_6.sInit.Description         :='Förderband Vereinzelner Wender GST';
ST03_461_B69_6.sInit.SensorType          :=sValveSensorType_WORK;

(* Init ST03_461_B69_7  ISK anwesend am Stopper (DigIn) *)
ST03_461_B69_7.sInit.InstName            :='ST03_461_B69_7';
ST03_461_B69_7.sInit.Description         :='ISK anwesend am Vereinzler';
ST03_461_B69_7.sInit.BitInName           :='+8-461_B69.7';
ST03_461_B69_7.sInit.HomePosSignal       :=2; (* 0: Signal=Low, 1: Signal=High, 2: always  *)
ST03_461_B69_7.sInit.MaxTime             :=2000;
ST03_461_B69_7.sInit.EnableInEveryMode   :=TRUE;

(* Init ST03_462_B70_0  Förderband  ISK anwesend Wender (DigIn) *)
ST03_462_B70_0.sInit.InstName            :='ST03_462_B70_0';
ST03_462_B70_0.sInit.Description         :='Förderband  ISK anwesend Wender';
ST03_462_B70_0.sInit.BitInName           :='+8-462_B70.0';
ST03_462_B70_0.sInit.HomePosSignal       :=2; (* 0: Signal=Low, 1: Signal=High, 2: always  *)
ST03_462_B70_0.sInit.MaxTime             :=2000;
ST03_462_B70_0.sInit.EnableInEveryMode   :=TRUE;

(* Init ST03_462_B70_1  Züführung  ISK Lageerkennung 1 (DigIn) *)
ST03_462_B70_1.sInit.InstName            :='ST03_462_B70_1';
ST03_462_B70_1.sInit.Description         :='Züführung  ISK Lageerkennung 1';
ST03_462_B70_1.sInit.BitInName           :='+8-462_B70.1';
ST03_462_B70_1.sInit.HomePosSignal       :=2; (* 0: Signal=Low, 1: Signal=High, 2: always  *)
ST03_462_B70_1.sInit.MaxTime             :=2000;
ST03_462_B70_1.sInit.EnableInEveryMode   :=TRUE;

(* Init ST03_462_B70_2  Züführung  ISK Lageerkennung 2 (DigIn) *)
ST03_462_B70_2.sInit.InstName            :='ST03_462_B70_2';
ST03_462_B70_2.sInit.Description         :='Züführung  ISK Lageerkennung 2';
ST03_462_B70_2.sInit.BitInName           :='+8-462_B70.2';
ST03_462_B70_2.sInit.HomePosSignal       :=2; (* 0: Signal=Low, 1: Signal=High, 2: always  *)
ST03_462_B70_2.sInit.MaxTime             :=2000;
ST03_462_B70_2.sInit.EnableInEveryMode   :=TRUE;

(* Init ST03_463_B70_3 Züführung  ISK Zylinder Vakuumdüsen AST (ValveSensor) *)
ST03_463_B70_3.sInit.InstName            :='ST03_463_B70_3';
ST03_463_B70_3.sInit.BitName            :='+8_463_B70.3';
ST03_463_B70_3.sInit.Description         :='Züführung  ISK Zylinder Vakuumdüsen AST';
ST03_463_B70_3.sInit.SensorType          :=sValveSensorType_INIT;

(* Init ST03_463_B70_4 Züführung  ISK Zylinder Vakuumdüsen GST (ValveSensor) *)
ST03_463_B70_4.sInit.InstName            :='ST03_463_B70_4';
ST03_463_B70_4.sInit.BitName            :='+8_463_B70.4';
ST03_463_B70_4.sInit.Description         :='Züführung  ISK Zylinder Vakuumdüsen GST';
ST03_463_B70_4.sInit.SensorType          :=sValveSensorType_WORK;

(* Init ST03_463_B70_5 Züführung  ISK Wendestation Einlauf (ValveSensor) *)
ST03_463_B70_5.sInit.InstName            :='ST03_463_B70_5';
ST03_463_B70_5.sInit.BitName            :='+8_463_B70.5';
ST03_463_B70_5.sInit.Description         :='Züführung  ISK Wendestation Einlauf AST';
ST03_463_B70_5.sInit.SensorType          :=sValveSensorType_INIT;

(* Init ST03_463_B70_6  Züführung  ISK Wendestation Auslauf (ValveSensor) *)
ST03_463_B70_6.sInit.InstName            :='ST03_463_B70_6';
ST03_463_B70_6.sInit.BitName            :='+8_463_B70.6';
ST03_463_B70_6.sInit.Description         :='Züführung  ISK Wendestation Auslauf GST';
ST03_463_B70_6.sInit.SensorType          :=sValveSensorType_WORK;

(* Init ST03_463_B70_7  ISK anwesend Übergabeposition Roboter (DigIn) *)
ST03_463_B70_7.sInit.InstName            :='ST03_463_B70_7';
ST03_463_B70_7.sInit.Description         :='Zuführung ISK auf Übergabeposition Robo Palettierer ';
ST03_463_B70_7.sInit.BitInName           :='+8-463_B70.4';
ST03_463_B70_7.sInit.HomePosSignal       :=2; (* 0: Signal=Low, 1: Signal=High, 2: always  *)
ST03_463_B70_7.sInit.MaxTime             :=2000;
ST03_463_B70_7.sInit.EnableInEveryMode   :=TRUE;

(* Init ST03_464_Y71_0  Förderband  Zuführung Vereinzelner Wender  (Valve) *)
ST03_464_Y71_0.sInit.InstName            :='ST03_464_Y71_0';
ST03_464_Y71_0.sInit.BitName            :='+8-464_Y71.0';
ST03_464_Y71_0.sInit.Description         :='Förderband  Zuführung Vereinzler Wender';
ST03_464_Y71_0.sInit.HomePosDefine       :=HOME_ALWAYS;
ST03_464_Y71_0.sInit.InitDescription     :='GS einfahren';
ST03_464_Y71_0.sInit.WorkDescription     :='AS ausfahren';
ST03_464_Y71_0.sInit.DampBothTime        :=200;
ST03_464_Y71_0.sInit.KindOfValve         :='A';
ST03_464_Y71_0.sInit.MaxTime             :=2000;

(* Init ST03_464_Y71_1  Förderband Zuführung Zylinder Vakuumdüsen (Valve) *)
ST03_464_Y71_1.sInit.InstName            :='ST03_464_Y71_1';
ST03_464_Y71_1.sInit.BitName            :='+8-464_Y71.1';
ST03_464_Y71_1.sInit.Description         :=' Förderband Zuführung Zylinder Vakuumdüsen';
ST03_464_Y71_1.sInit.HomePosDefine       :=HOME_ALWAYS;
ST03_464_Y71_1.sInit.InitDescription     :='GS einfahren';
ST03_464_Y71_1.sInit.WorkDescription     :='AS ausfahren';
ST03_464_Y71_1.sInit.DampBothTime        :=200;
ST03_464_Y71_1.sInit.KindOfValve         :='A';
ST03_464_Y71_1.sInit.MaxTime             :=2000;

(* Init ST03_464_Y71_2  Förderband  Zuführung Wendestation  (Valve) *)
ST03_464_Y71_2.sInit.InstName            :='ST03_464_Y71_2';
ST03_464_Y71_2.sInit.BitName            :='+8-464_Y71.2';
ST03_464_Y71_2.sInit.Description         :='Förderband  Zuführung Wendestation';
ST03_464_Y71_2.sInit.HomePosDefine       :=HOME_ALWAYS;
ST03_464_Y71_2.sInit.InitDescription     :='IN';
ST03_464_Y71_2.sInit.WorkDescription     :='OUT';
ST03_464_Y71_2.sInit.DampBothTime        :=200;
ST03_464_Y71_2.sInit.KindOfValve         :='A';
ST03_464_Y71_2.sInit.MaxTime             :=2000;

(* Init ST03_464_Y71_3 Förderband  Zuführung Vereinzler (Valve) *)
ST03_464_Y71_3.sInit.InstName            :='ST03_464_Y71_3';
ST03_464_Y71_3.sInit.BitName            :='+8-464_Y71.3';
ST03_464_Y71_3.sInit.Description         :='Förderband  Zuführung Vereinzler';
ST03_464_Y71_3.sInit.HomePosDefine       :=HOME_ALWAYS;
ST03_464_Y71_3.sInit.InitDescription     :='GS einfahren';
ST03_464_Y71_3.sInit.WorkDescription     :='AS ausfahren';
ST03_464_Y71_3.sInit.DampBothTime        :=200;
ST03_464_Y71_3.sInit.KindOfValve         :='A';
ST03_464_Y71_3.sInit.MaxTime             :=2000;

(* Init ST03_464_Y71_4 Förderband  Zuführung Stopper (Valve) *)
ST03_464_Y71_4.sInit.InstName            :='ST03_464_Y71_4';
ST03_464_Y71_4.sInit.BitName            :='+8-464_Y71.4';
ST03_464_Y71_4.sInit.Description         :='Förderband  Zuführung Stopper';
ST03_464_Y71_4.sInit.HomePosDefine       :=HOME_ALWAYS;
ST03_464_Y71_4.sInit.InitDescription     :='GS ausfahren';
ST03_464_Y71_4.sInit.WorkDescription     :='AS einfahren';
ST03_464_Y71_4.sInit.DampBothTime        :=200;
ST03_464_Y71_4.sInit.KindOfValve         :='A';
ST03_464_Y71_4.sInit.MaxTime             :=2000;

(* Init ST03_464_Y71_5 Vakuumdüse ein/aus (Valve) *)
ST03_464_Y71_5.sInit.InstName            :='ST03_464_Y71_5';
ST03_464_Y71_5.sInit.BitName            :='+8-464_Y71.5';
ST03_464_Y71_5.sInit.Description         :='Vakuumdüse ein/aus';
ST03_464_Y71_5.sInit.HomePosDefine       :=HOME_ALWAYS;
ST03_464_Y71_5.sInit.InitDescription     :='OFF';
ST03_464_Y71_5.sInit.WorkDescription     :='ON';
ST03_464_Y71_5.sInit.DampBothTime        :=200;
ST03_464_Y71_5.sInit.KindOfValve         :='A';
ST03_464_Y71_5.sInit.MaxTime             :=2000;

(* Init ST03_464_B71_6  Vakum vorhanden (DigIn) *)
ST03_464_B71_6.sInit.InstName            :='ST03_464_B71_6';
ST03_464_B71_6.sInit.Description         :='Vakum vorhanden ';
ST03_464_B71_6.sInit.BitInName           :='+8-464_B71.6';
ST03_464_B71_6.sInit.HomePosSignal       :=2; (* 0: Signal=Low, 1: Signal=High, 2: always  *)
ST03_464_B71_6.sInit.MaxTime             :=2000;
ST03_464_B71_6.sInit.EnableInEveryMode   :=TRUE;

(* Init ST03_464_B71_7 Förderband Staustrecke mitte voll (DigIn) *)
ST03_464_B71_7.sInit.InstName            :='ST03_464_B71_7';
ST03_464_B71_7.sInit.Description         :='Staustrecke mitte voll ';
ST03_464_B71_7.sInit.BitInName           :='+8-464_B71.7';
ST03_464_B71_7.sInit.HomePosSignal       :=2; (* 0: Signal=Low, 1: Signal=High, 2: always  *)
ST03_464_B71_7.sInit.MaxTime             :=2000;
ST03_464_B71_7.sInit.EnableInEveryMode   :=TRUE;
END_ACTION
ACTION Init_48pol:
(*Rüstsatz 48 pol ==================================================================================*)

(* Init ST03_551_B69_0 Zuführung  frei zum Ablegen ISK SP Maschine (DigIn) *)
ST03_551_B69_0.sInit.InstName            :='ST03_551_B69_0';
ST03_551_B69_0.sInit.Description         :='frei zum Ablegen ISK SP Maschine';
ST03_551_B69_0.sInit.BitInName           :='+8-551_B69.0';
ST03_551_B69_0.sInit.HomePosSignal       :=2; (* 0: Signal=Low, 1: Signal=High, 2: always  *)
ST03_551_B69_0.sInit.MaxTime             :=2000;
ST03_551_B69_0.sInit.EnableInEveryMode   :=TRUE;

(* Init ST03_551_B69_1 Zuführung Vereinzler eingefahren GST (ValveSensor) *)
ST03_551_B69_1.sInit.InstName		:='ST03_551_B69_1';
ST03_551_B69_1.sInit.BitName		:='+8_551_B69.1';
ST03_551_B69_1.sInit.Description	:=' Vereinzler eingefahren GST';
ST03_551_B69_1.sInit.SensorType	:=sValveSensorType_INIT;

(* Init ST03_551_B69_2 Zuführung Vereinzler ausgefahren AST (ValveSensor) *)
ST03_551_B69_2.sInit.InstName		:='ST03_551_B69_2';
ST03_551_B69_2.sInit.BitName		:='+8_551_B69.2';
ST03_551_B69_2.sInit.Description	:=' Vereinzler ausgefahren AST';
ST03_551_B69_2.sInit.SensorType	:=sValveSensorType_WORK;

(* Init ST03_551_B69_3 Zuführung Stopper eingefahren AST (ValveSensor) *)
ST03_551_B69_3.sInit.InstName		:='ST03_551_B69_3';
ST03_551_B69_3.sInit.BitName		:='+8_551_B69.3';
ST03_551_B69_3.sInit.Description	:='Stopper eingefahren AST';
ST03_551_B69_3.sInit.SensorType	:=sValveSensorType_WORK;

(* Init ST03_551_B69_4 Zuführung Stopper ausgefahren GST (ValveSensor) *)
ST03_551_B69_4.sInit.InstName		:='ST03_551_B69_4';
ST03_551_B69_4.sInit.BitName		:='+8_551_B69.4';
ST03_551_B69_4.sInit.Description	:='Stopper ausgefahren GST';
ST03_551_B69_4.sInit.SensorType	:=sValveSensorType_INIT;;

(* Init ST03_551_B69_6 ISK anwesend am Stopper (DigIn) *)
ST03_551_B69_6.sInit.InstName            :='ST03_551_B69_6';
ST03_551_B69_6.sInit.Description         :='ISK anwesend am Stopper';
ST03_551_B69_6.sInit.BitInName           :='+8-551_B69.6';
ST03_551_B69_6.sInit.HomePosSignal       :=2; (* 0: Signal=Low, 1: Signal=High, 2: always  *)
ST03_551_B69_6.sInit.MaxTime             :=2000;
ST03_551_B69_6.sInit.EnableInEveryMode   :=TRUE;

(* Init ST03_551_B69_7 ISK rechts Lageerkennung (DigIn) *)
ST03_551_B69_7.sInit.InstName            :='ST03_551_B69_7';
ST03_551_B69_7.sInit.Description         :='ISK rechts Lageerkennung.';
ST03_551_B69_7.sInit.BitInName           :='+8-551_B69.7';
ST03_551_B69_7.sInit.HomePosSignal       :=2; (* 0: Signal=Low, 1: Signal=High, 2: always  *)
ST03_551_B69_7.sInit.MaxTime             :=2000;
ST03_551_B69_7.sInit.EnableInEveryMode   :=TRUE;

(* Init ST03_552_B70_0 ISK links Lageerkennung (DigIn) *)
ST03_552_B70_0.sInit.InstName            :='ST03_552_B70_0';
ST03_552_B70_0.sInit.Description         :='ISK links Lageerkennung';
ST03_552_B70_0.sInit.BitInName           :='+8-552_B70.0';
ST03_552_B70_0.sInit.HomePosSignal       :=2; (* 0: Signal=Low, 1: Signal=High, 2: always  *)
ST03_552_B70_0.sInit.MaxTime             :=2000;
ST03_552_B70_0.sInit.EnableInEveryMode   :=TRUE;

(* Init ST03_552_Y70_1   Zuführung  Vereinzler AST/GST (Valve) *)
ST03_552_Y70_1.sInit.InstName            :='ST03_552_Y70_1';
ST03_552_Y70_1.sInit.BitName            :='+8-552_Y70.1';
ST03_552_Y70_1.sInit.Description         :=' Zuführung Vereinzler AST/GST';
ST03_552_Y70_1.sInit.HomePosDefine       :=HOME_ALWAYS;
ST03_552_Y70_1.sInit.InitDescription     :='GS einfahren';
ST03_552_Y70_1.sInit.WorkDescription     :='AS ausfahren';
ST03_552_Y70_1.sInit.DampBothTime        :=200;
ST03_552_Y70_1.sInit.KindOfValve         :='A';
ST03_552_Y70_1.sInit.MaxTime             :=2000;

(* Init ST03_552_Y70_2   Zuführung  Stopper AST/GST (Valve) *)
ST03_552_Y70_2.sInit.InstName            :='ST03_552_Y70_2';
ST03_552_Y70_2.sInit.BitName            :='+8-552_Y70.2';
ST03_552_Y70_2.sInit.Description         :=' Zuführung Stopper AST/GST';
ST03_552_Y70_2.sInit.HomePosDefine       :=HOME_ALWAYS;
ST03_552_Y70_2.sInit.InitDescription     :='GS ausfahren';
ST03_552_Y70_2.sInit.WorkDescription     :='AS einfahren';
ST03_552_Y70_2.sInit.DampBothTime        :=200;
ST03_552_Y70_2.sInit.KindOfValve         :='A';
ST03_552_Y70_2.sInit.MaxTime             :=2000;
END_ACTION
ACTION Init_72pol:
(*Rüstsatz 72 pol ==================================================================================*)

(* Init ST03_546_B69_0 Zuführung  frei zum Ablegen ISK SP Maschine (DigIn) *)
ST03_546_B69_0.sInit.InstName            :='ST03_546_B69_0';
ST03_546_B69_0.sInit.Description         :='frei zum Ablegen ISK SP Maschine';
ST03_546_B69_0.sInit.BitInName           :='+8-546_B69.0';
ST03_546_B69_0.sInit.HomePosSignal       :=2; (* 0: Signal=Low, 1: Signal=High, 2: always  *)
ST03_546_B69_0.sInit.MaxTime             :=2000;
ST03_546_B69_0.sInit.EnableInEveryMode   :=TRUE;

(* Init ST03_546_B69_1 Zuführung Vereinzler eingefahren GST (ValveSensor) *)
ST03_546_B69_1.sInit.InstName		:='ST03_546_B69_1';
ST03_546_B69_1.sInit.BitName		:='+8_546_B69.1';
ST03_546_B69_1.sInit.Description	:=' Vereinzler eingefahren GST';
ST03_546_B69_1.sInit.SensorType	:=sValveSensorType_INIT;

(* Init ST03_546_B69_2 Zuführung Vereinzler ausgefahren AST (ValveSensor) *)
ST03_546_B69_2.sInit.InstName		:='ST03_546_B69_2';
ST03_546_B69_2.sInit.BitName		:='+8_546_B69.2';
ST03_546_B69_2.sInit.Description	:=' Vereinzler ausgefahren AST';
ST03_546_B69_2.sInit.SensorType	:=sValveSensorType_WORK;

(* Init ST03_546_B69_3 Zuführung Stopper eingefahren AST (ValveSensor) *)
ST03_546_B69_3.sInit.InstName		:='ST03_546_B69_3';
ST03_546_B69_3.sInit.BitName		:='+8_546_B69.3';
ST03_546_B69_3.sInit.Description	:='Stopper eingefahren AST';
ST03_546_B69_3.sInit.SensorType	:=sValveSensorType_WORK;

(* Init ST03_546_B69_4 Zuführung Stopper ausgefahren GST (ValveSensor) *)
ST03_546_B69_4.sInit.InstName		:='ST03_546_B69_4';
ST03_546_B69_4.sInit.BitName		:='+8_546_B69.4';
ST03_546_B69_4.sInit.Description	:='Stopper ausgefahren GST';
ST03_546_B69_4.sInit.SensorType	:=sValveSensorType_INIT;;

(* Init ST03_546_B69_6 ISK anwesend am Stopper (DigIn) *)
ST03_546_B69_6.sInit.InstName            :='ST03_546_B69_6';
ST03_546_B69_6.sInit.Description         :='ISK anwesend am Stopper';
ST03_546_B69_6.sInit.BitInName           :='+8-546_B69.6';
ST03_546_B69_6.sInit.HomePosSignal       :=2; (* 0: Signal=Low, 1: Signal=High, 2: always  *)
ST03_546_B69_6.sInit.MaxTime             :=2000;
ST03_546_B69_6.sInit.EnableInEveryMode   :=TRUE;

(* Init ST03_546_B69_7 ISK rechts Lageerkennung (DigIn) *)
ST03_546_B69_7.sInit.InstName            :='ST03_546_B69_7';
ST03_546_B69_7.sInit.Description         :='ISK rechts Lageerkennung.';
ST03_546_B69_7.sInit.BitInName           :='+8-546_B69.7';
ST03_546_B69_7.sInit.HomePosSignal       :=2; (* 0: Signal=Low, 1: Signal=High, 2: always  *)
ST03_546_B69_7.sInit.MaxTime             :=2000;
ST03_546_B69_7.sInit.EnableInEveryMode   :=TRUE;

(* Init ST03_547_B70_0 ISK links Lageerkennung (DigIn) *)
ST03_547_B70_0.sInit.InstName            :='ST03_547_B70_0';
ST03_547_B70_0.sInit.Description         :='ISK links Lageerkennung';
ST03_547_B70_0.sInit.BitInName           :='+8-547_B70.0';
ST03_547_B70_0.sInit.HomePosSignal       :=2; (* 0: Signal=Low, 1: Signal=High, 2: always  *)
ST03_547_B70_0.sInit.MaxTime             :=2000;
ST03_547_B70_0.sInit.EnableInEveryMode   :=TRUE;

(* Init ST03_547_Y70_1   Zuführung  Vereinzler AST/GST (Valve) *)
ST03_547_Y70_1.sInit.InstName            :='ST03_547_Y70_1';
ST03_547_Y70_1.sInit.BitName            :='+8-547_Y70.1';
ST03_547_Y70_1.sInit.Description         :='Zuführung Vereinzler AST/GST';
ST03_547_Y70_1.sInit.HomePosDefine       :=HOME_ALWAYS;
ST03_547_Y70_1.sInit.InitDescription     :='GS einfahren';
ST03_547_Y70_1.sInit.WorkDescription     :='AS ausfahren';
ST03_547_Y70_1.sInit.DampBothTime        :=200;
ST03_547_Y70_1.sInit.KindOfValve         :='A';
ST03_547_Y70_1.sInit.MaxTime             :=2000;

(* Init ST03_547_Y70_2   Zuführung  Stopper AST/GST (Valve) *)
ST03_547_Y70_2.sInit.InstName            :='ST03_547_Y70_2';
ST03_547_Y70_2.sInit.BitName            :='+8-547_Y70.2';
ST03_547_Y70_2.sInit.Description         :='Zuführung Stopper AST/GST';
ST03_547_Y70_2.sInit.HomePosDefine       :=HOME_ALWAYS;
ST03_547_Y70_2.sInit.InitDescription     :='GS ausfahren';
ST03_547_Y70_2.sInit.WorkDescription     :='AS einfahren';
ST03_547_Y70_2.sInit.DampBothTime        :=200;
ST03_547_Y70_2.sInit.KindOfValve         :='A';
ST03_547_Y70_2.sInit.MaxTime             :=2000;
END_ACTION
ACTION Init_7pol:
(*Rüstsatz 7 pol==================================================================================*)

(* Init ST03_512_XG1 ISK in Klemmer (DigIn) *)
ST03_512_XG1.sInit.InstName            :='ST03_512_XG1';
ST03_512_XG1.sInit.Description         :='ISK in Klemmer';
ST03_512_XG1.sInit.BitInName           :='+8-512_XG1';
ST03_512_XG1.sInit.HomePosSignal       :=2; (* 0: Signal=Low, 1: Signal=High, 2: always  *)
ST03_512_XG1.sInit.MaxTime             :=2000;
ST03_512_XG1.sInit.EnableInEveryMode   :=TRUE;

(* Init ST03_512_B69_1 ISK Klemmer 1 AST (ValveSensor) *)
ST03_512_B69_1.sInit.InstName		:='ST03_512_B69_1';
ST03_512_B69_1.sInit.BitName		:='+8_512_B69.1';
ST03_512_B69_1.sInit.Description	:='ISK Klemmer 1 AST';
ST03_512_B69_1.sInit.SensorType	:=sValveSensorType_WORK;

(* Init ST03_512_B69_2 ISK Klemmer 1 GST (ValveSensor) *)
ST03_512_B69_2.sInit.InstName		:='ST03_512_B69_2';
ST03_512_B69_2.sInit.BitName		:='+8_512_B69.2';
ST03_512_B69_2.sInit.Description	:='ISK Klemmer 1 GST';
ST03_512_B69_2.sInit.SensorType	:=sValveSensorType_INIT;

(* Init ST03_512_B69_3 ISK Klemmer 1 AST (ValveSensor) *)
ST03_512_B69_3.sInit.InstName		:='ST03_512_B69_3';
ST03_512_B69_3.sInit.BitName		:='+8_512_B69.3';
ST03_512_B69_3.sInit.Description	:='ISK Klemmer 2 AST';
ST03_512_B69_3.sInit.SensorType	:=sValveSensorType_WORK;

(* Init ST03_512_B69_4 ISK Klemmer 1 GST (ValveSensor) *)
ST03_512_B69_4.sInit.InstName		:='ST03_512_B69_4';
ST03_512_B69_4.sInit.BitName		:='+8_512_B69.4';
ST03_512_B69_4.sInit.Description	:='ISK Klemmer 2 GST';
ST03_512_B69_4.sInit.SensorType	:=sValveSensorType_INIT;

(* Init ST03_512_B69_5 Rinne schwenkern 0° AST (ValveSensor) *)
ST03_512_B69_5.sInit.InstName		:='ST03_512_B69_5';
ST03_512_B69_5.sInit.BitName		:='+8_512_B69.5';
ST03_512_B69_5.sInit.Description	:='Rinne schwenkern 0° AST';
ST03_512_B69_5.sInit.SensorType	:=sValveSensorType_WORK;

(* Init ST03_512_B69_6 Rinne schwenkern 180° GST (ValveSensor) *)
ST03_512_B69_6.sInit.InstName		:='ST03_512_B69_6';
ST03_512_B69_6.sInit.BitName		:='+8_512_B69.6';
ST03_512_B69_6.sInit.Description	:='Rinne schwenkern 180° GST';
ST03_512_B69_6.sInit.SensorType	:=sValveSensorType_INIT;

(* Init ST03_513_B70_0 Führungsschiene  Zuführung Vereinzler AST (ValveSensor) *)
ST03_513_B70_0.sInit.InstName		:='ST03_513_B70_0';
ST03_513_B70_0.sInit.BitName		:='+8_513_B70.0';
ST03_513_B70_0.sInit.Description	:='Führungsschiene  Zuführung Vereinzler AST';
ST03_513_B70_0.sInit.SensorType	:=sValveSensorType_WORK;

(* Init ST03_513_B70_1 Führungsschiene  Zuführung Vereinzler GST (ValveSensor) *)
ST03_513_B70_1.sInit.InstName		:='ST03_513_B70_1';
ST03_513_B70_1.sInit.BitName		:='+8_513_B70.1';
ST03_513_B70_1.sInit.Description	:='Führungsschiene  Zuführung Vereinzler GST';
ST03_513_B70_1.sInit.SensorType	:=sValveSensorType_INIT;

